(* IEC 61131-3 sources: PLC_02/HMI (part 2) *)

	IF (HMI.Rack4[13] AND 16#00ff) >= 1 AND (HMI.Rack4[13] AND 16#00ff) <= 164 THEN
		HMIBinding.CommonUI.sString5[0]		:= UINT_TO_STRING((HMI.Rack4[13] AND 16#00ff)) ;
	ELSIF (HMI.Rack4[13] AND 16#00ff) < 1 THEN
		HMIBinding.CommonUI.sString5[0]		:= '1';
	ELSE
		HMIBinding.CommonUI.sString5[0]		:= '164';
	END_IF;
	IF (HMI.Rack4[13]  /  16#0100) >= 1 AND (HMI.Rack4[13]  /  16#0100) <= 164 THEN
		HMIBinding.CommonUI.sString5[1] 		:= UINT_TO_STRING(HMI.Rack4[13]  /  16#0100) ;
	ELSIF (HMI.Rack4[13]  /  16#0100) < 1 THEN
		HMIBinding.CommonUI.sString5[1]		:= '1';
	ELSE
		HMIBinding.CommonUI.sString5[1]		:= '164';
	END_IF;
	HMIBinding.CommonUI.sString20[5]		:= CONCAT(HMIBinding.CommonUI.sString5[0],'(C)');
	HMIBinding.CommonUI.sString20[6]		:= CONCAT(HMIBinding.CommonUI.sString5[1],'(C)');

	IF (HMI.Rack4[14] AND 16#00ff) >= 1 AND (HMI.Rack4[14] AND 16#00ff) <= 164 THEN
		HMIBinding.CommonUI.sString5[0]		:= UINT_TO_STRING((HMI.Rack4[14] AND 16#00ff)) ;
	ELSIF (HMI.Rack4[14] AND 16#00ff) < 1 THEN
		HMIBinding.CommonUI.sString5[0]		:= '1';
	ELSE
		HMIBinding.CommonUI.sString5[0]		:= '164';
	END_IF;
	IF (HMI.Rack4[14]  /  16#0100) >= 1 AND (HMI.Rack4[14]  /  16#0100) <= 164 THEN
		HMIBinding.CommonUI.sString5[1] 		:= UINT_TO_STRING(HMI.Rack4[14]  /  16#0100) ;
	ELSIF (HMI.Rack4[14]  /  16#0100) < 1 THEN
		HMIBinding.CommonUI.sString5[1]		:= '1';
	ELSE
		HMIBinding.CommonUI.sString5[1]		:= '164';
	END_IF;
	HMIBinding.CommonUI.sString20[7]		:= CONCAT(HMIBinding.CommonUI.sString5[0],'(C)');
	HMIBinding.CommonUI.sString20[8]		:= CONCAT(HMIBinding.CommonUI.sString5[1],'(C)');

	IF HMI.Rack4[22] >= 672 AND HMI.Rack4[22] <= 1080 THEN
		HMIBinding.RackUI.sString5[0] 	:= REAL_TO_STRING(HMI.Rack4[22]*0.1) ;
	ELSIF HMI.Rack4[22] < 672 THEN
		HMIBinding.RackUI.sString5[0]	:= '67.2';
	ELSE
		HMIBinding.RackUI.sString5[0]	:= '108';
	END_IF;
	HMIBinding.RackUI.sString20[1]		:= CONCAT(HMIBinding.RackUI.sString5[0],'(V)');

	IF (HMI.Rack4[21].0) THEN
		HMIBinding.RackUI.sString20[0] := 'Solid_Green';
	ELSE
		HMIBinding.RackUI.sString20[0] := 'Solid_Red';
	END_IF;
	IF HMI.Rack4[23] >= 672 AND HMI.Rack4[23] <= 1080 THEN
		HMIBinding.RackUI.sString5[0] 	:= REAL_TO_STRING(HMI.Rack4[23]*0.1) ;
	ELSIF HMI.Rack4[23] < 672 THEN
		HMIBinding.RackUI.sString5[0]	:= '67.2';
	ELSE
		HMIBinding.RackUI.sString5[0]	:= '108';
	END_IF;
	HMIBinding.RackUI.sString20[3]		:= CONCAT(HMIBinding.RackUI.sString5[0],'(V)');

	IF (HMI.Rack4[21].1) THEN
		HMIBinding.RackUI.sString20[2] := 'Solid_Green';
	ELSE
		HMIBinding.RackUI.sString20[2] := 'Solid_Red';
	END_IF;

	IF HMI.Rack4[24] >= 672 AND HMI.Rack4[24] <= 1080 THEN
		HMIBinding.RackUI.sString5[0] 	:= REAL_TO_STRING(HMI.Rack4[24]*0.1) ;
	ELSIF HMI.Rack4[24] < 672 THEN
		HMIBinding.RackUI.sString5[0]	:= '67.2';
	ELSE
		HMIBinding.RackUI.sString5[0]	:= '108';
	END_IF;
	HMIBinding.RackUI.sString20[5]		:= CONCAT(HMIBinding.RackUI.sString5[0],'(V)');

	IF (HMI.Rack4[21].2) THEN
		HMIBinding.RackUI.sString20[4] := 'Solid_Green';
	ELSE
		HMIBinding.RackUI.sString20[4] := 'Solid_Red';
	END_IF;

	IF HMI.Rack4[25] >= 672 AND HMI.Rack4[25] <= 1080 THEN
		HMIBinding.RackUI.sString5[0] 	:= REAL_TO_STRING(HMI.Rack4[25]*0.1) ;
	ELSIF HMI.Rack4[25] < 672 THEN
		HMIBinding.RackUI.sString5[0]	:= '67.2';
	ELSE
		HMIBinding.RackUI.sString5[0]	:= '108';
	END_IF;
	HMIBinding.RackUI.sString20[7]		:= CONCAT(HMIBinding.RackUI.sString5[0],'(V)');

	IF (HMI.Rack4[21].3) THEN
		HMIBinding.RackUI.sString20[6] := 'Solid_Green';
	ELSE
		HMIBinding.RackUI.sString20[6] := 'Solid_Red';
	END_IF;
	IF HMI.Rack4[26] >= 672 AND HMI.Rack4[26] <= 1080 THEN
		HMIBinding.RackUI.sString5[0] 	:= REAL_TO_STRING(HMI.Rack4[26]*0.1) ;
	ELSIF HMI.Rack4[26] < 672 THEN
		HMIBinding.RackUI.sString5[0]	:= '67.2';
	ELSE
		HMIBinding.RackUI.sString5[0]	:= '108';
	END_IF;
	HMIBinding.RackUI.sString20[9]		:= CONCAT(HMIBinding.RackUI.sString5[0],'(V)');

	IF (HMI.Rack4[21].4) THEN
		HMIBinding.RackUI.sString20[8] := 'Solid_Green';
	ELSE
		HMIBinding.RackUI.sString20[8] := 'Solid_Red';
	END_IF;
	IF HMI.Rack4[27] >= 672 AND HMI.Rack4[27] <= 1080 THEN
		HMIBinding.RackUI.sString5[0] 	:= REAL_TO_STRING(HMI.Rack4[27]*0.1) ;
	ELSIF HMI.Rack4[27] < 672 THEN
		HMIBinding.RackUI.sString5[0]	:= '67.2';
	ELSE
		HMIBinding.RackUI.sString5[0]	:= '108';
	END_IF;
	HMIBinding.RackUI.sString20[11]		:= CONCAT(HMIBinding.RackUI.sString5[0],'(V)');

	IF (HMI.Rack4[21].5) THEN
		HMIBinding.RackUI.sString20[10] := 'Solid_Green';
	ELSE
		HMIBinding.RackUI.sString20[10] := 'Solid_Red';
	END_IF;
	IF HMI.Rack4[28] >= 672 AND HMI.Rack4[28] <= 1080 THEN
		HMIBinding.RackUI.sString5[0] 	:= REAL_TO_STRING(HMI.Rack4[28]*0.1) ;
	ELSIF HMI.Rack4[28] < 672 THEN
		HMIBinding.RackUI.sString5[0]	:= '67.2';
	ELSE
		HMIBinding.RackUI.sString5[0]	:= '108';
	END_IF;
	HMIBinding.RackUI.sString20[13]		:= CONCAT(HMIBinding.RackUI.sString5[0],'(V)');

	IF (HMI.Rack4[21].6) THEN
		HMIBinding.RackUI.sString20[12] := 'Solid_Green';
	ELSE
		HMIBinding.RackUI.sString20[12] := 'Solid_Red';
	END_IF;

	(* Over Current *)
	IF HMI.Rack4[17].0 THEN
		HMIBinding.RackUI.sString20[14] 		:= 'Solid_Red';
	ELSIF HMI.Rack4[16].0 THEN
		HMIBinding.RackUI.sString20[14]			:= 'Solid_Orange';
	ELSIF HMI.Rack4[15].0 THEN
		HMIBinding.RackUI.sString20[14]			:= 'Solid_Yellow';
	ELSE
		HMIBinding.RackUI.sString20[14]			:= 'Solid_Green';
	END_IF;

	(* Over SOC *)
	IF HMI.Rack4[17].1 THEN
		HMIBinding.RackUI.sString20[15]			:= 'Solid_Red';
	ELSIF HMI.Rack4[16].1 THEN
		HMIBinding.RackUI.sString20[15]			:= 'Solid_Orange';
	ELSIF HMI.Rack4[15].1 THEN
		HMIBinding.RackUI.sString20[15]			:= 'Solid_Yellow';
	ELSE
		HMIBinding.RackUI.sString20[15] 			:= 'Solid_Green';
	END_IF;

	(* Under SOC *)
	IF HMI.Rack4[17].2 THEN
		HMIBinding.RackUI.sString20[16] 			:= 'Solid_Red';
	ELSIF HMI.Rack4[16].2 THEN
		HMIBinding.RackUI.sString20[16]  			:= 'Solid_Orange';
	ELSIF HMI.Rack4[15].2 THEN
		HMIBinding.RackUI.sString20[16] 			:= 'Solid_Yellow';
	ELSE
		HMIBinding.RackUI.sString20[16]			:= 'Solid_Green';
	END_IF;

	(* Over Voltage *)
	IF HMI.Rack4[17].3 THEN
		HMIBinding.RackUI.sString20[17]			:= 'Solid_Red';
	ELSIF HMI.Rack4[16].3 THEN
		HMIBinding.RackUI.sString20[17] 			:= 'Solid_Orange';
	ELSIF HMI.Rack4[15].3 THEN
		HMIBinding.RackUI.sString20[17] 			:= 'Solid_Yellow';
	ELSE
		HMIBinding.RackUI.sString20[17] 			:= 'Solid_Green';
	END_IF;

	(* Under Voltage *)
	IF HMI.Rack4[17].4 THEN
		HMIBinding.RackUI.sString20[18] 			:= 'Solid_Red';
	ELSIF HMI.Rack4[16].4 THEN
		HMIBinding.RackUI.sString20[18] 			:= 'Solid_Orange';
	ELSIF HMI.Rack4[15].4 THEN
		HMIBinding.RackUI.sString20[18] 			:= 'Solid_Yellow';
	ELSE
		HMIBinding.RackUI.sString20[18] 			:= 'Solid_Green';
	END_IF;

	(* Cell Over Voltage *)
	IF HMI.Rack4[17].5 THEN
		HMIBinding.RackUI.sString20[19] 			:= 'Solid_Red';
	ELSIF HMI.Rack4[16].5 THEN
		HMIBinding.RackUI.sString20[19] 			:= 'Solid_Orange';
	ELSIF HMI.Rack4[15].5 THEN
		HMIBinding.RackUI.sString20[19] 			:= 'Solid_Yellow';
	ELSE
		HMIBinding.RackUI.sString20[19] 			:= 'Solid_Green';
	END_IF;

	(* Cell Under Voltage *)
	IF HMI.Rack4[17].6 THEN
		HMIBinding.RackUI.sString20[20] 			:= 'Solid_Red';
	ELSIF HMI.Rack4[16].6 THEN
		HMIBinding.RackUI.sString20[20] 			:= 'Solid_Orange';
	ELSIF HMI.Rack4[15].6 THEN
		HMIBinding.RackUI.sString20[20] 			:= 'Solid_Yellow';
	ELSE
		HMIBinding.RackUI.sString20[20] 			:= 'Solid_Green';
	END_IF;

	(* Cell UnBalance Voltage *)
	IF HMI.Rack4[17].7 THEN
		HMIBinding.RackUI.sString20[21]			:= 'Solid_Red';
	ELSIF HMI.Rack4[16].7 THEN
		HMIBinding.RackUI.sString20[21] 			:= 'Solid_Orange';
	ELSIF HMI.Rack4[15].7 THEN
		HMIBinding.RackUI.sString20[21]			:= 'Solid_Yellow';
	ELSE
		HMIBinding.RackUI.sString20[21]			:= 'Solid_Green';
	END_IF;

	(* Discahrger Cell Over Temperature *)
	IF HMI.Rack4[17].8 THEN
		HMIBinding.RackUI.sString20[22] 			:= 'Solid_Red';
	ELSIF HMI.Rack4[16].8 THEN
		HMIBinding.RackUI.sString20[22] 			:= 'Solid_Orange';
	ELSIF HMI.Rack4[15].8 THEN
		HMIBinding.RackUI.sString20[22] 			:= 'Solid_Yellow';
	ELSE
		HMIBinding.RackUI.sString20[22] 			:= 'Solid_Green';
	END_IF;

	(* Charger Cell Over Temperature *)
	IF HMI.Rack4[17].9 THEN
		HMIBinding.RackUI.sString20[23] 			:= 'Solid_Red';
	ELSIF HMI.Rack4[16].9 THEN
		HMIBinding.RackUI.sString20[23] 			:= 'Solid_Orange';
	ELSIF HMI.Rack4[15].9 THEN
		HMIBinding.RackUI.sString20[23] 			:= 'Solid_Yellow';
	ELSE
		HMIBinding.RackUI.sString20[23] 			:= 'Solid_Green';
	END_IF;

	(* Discahrger Cell Under Temperature *)
	IF HMI.Rack4[17].10 THEN
		HMIBinding.RackUI.sString20[24] 			:= 'Solid_Red';
	ELSIF HMI.Rack4[16].10 THEN
		HMIBinding.RackUI.sString20[24] 			:= 'Solid_Orange';
	ELSIF HMI.Rack4[15].10 THEN
		HMIBinding.RackUI.sString20[24] 			:= 'Solid_Yellow';
	ELSE
		HMIBinding.RackUI.sString20[24] 			:= 'Solid_Green';
	END_IF;

	(* Charger Cell Under Temperature *)
	IF HMI.Rack4[17].11 THEN
		HMIBinding.RackUI.sString20[25] 		:= 'Solid_Red';
	ELSIF HMI.Rack4[16].11 THEN
		HMIBinding.RackUI.sString20[25]			:= 'Solid_Orange';
	ELSIF HMI.Rack4[15].11 THEN
		HMIBinding.RackUI.sString20[25]			:= 'Solid_Yellow';
	ELSE
		HMIBinding.RackUI.sString20[25]			:= 'Solid_Green';
	END_IF;

	(* Cell UnBalance Temperature *)
	IF HMI.Rack4[17].12 THEN
		HMIBinding.RackUI.sString20[26] 		:= 'Solid_Red';
	ELSIF HMI.Rack4[16].12 THEN
		HMIBinding.RackUI.sString20[26]			:= 'Solid_Orange';
	ELSIF HMI.Rack4[15].12 THEN
		HMIBinding.RackUI.sString20[26]			:= 'Solid_Yellow';
	ELSE
		HMIBinding.RackUI.sString20[26]			:= 'Solid_Green';
	END_IF;

	(* Internal COM *)
	IF HMI.Rack4[17].15 THEN
		HMIBinding.RackUI.sString20[27] 		:= 'Solid_Red';
	ELSE
		HMIBinding.RackUI.sString20[27]			:= 'Solid_Green';
	END_IF;

	(* External COM *)
	IF HMI.Rack4[17].0 THEN
		HMIBinding.RackUI.sString20[28] 		:= 'Solid_Red';
	ELSE
		HMIBinding.RackUI.sString20[28]			:= 'Solid_Green';
	END_IF;

	(* RelayWelding *)
	IF HMI.Rack4[18].1 THEN
		HMIBinding.RackUI.sString20[29] 		:= 'Solid_Red';
	ELSE
		HMIBinding.RackUI.sString20[29]			:= 'Solid_Green';
	END_IF;

	(* WaterLeak *)
	IF HMI.Rack4[18].2 THEN
		HMIBinding.RackUI.sString20[30] 		:= 'Solid_Red';
	ELSE
		HMIBinding.RackUI.sString20[30]			:= 'Solid_Green';
	END_IF;

	(* InsulationRegister *)
	IF HMI.Rack4[18].3 THEN
		HMIBinding.RackUI.sString20[31] 		:= 'Solid_Red';
	ELSE
		HMIBinding.RackUI.sString20[31]			:= 'Solid_Green';
	END_IF;

	(* MDSFuse *)
	IF HMI.Rack4[18].4 THEN
		HMIBinding.RackUI.sString20[32] 		:= 'Solid_Red';
	ELSE
		HMIBinding.RackUI.sString20[32]			:= 'Solid_Green';
	END_IF;

	(* CoolingRack *)
	IF HMI.Rack4[18].5 THEN
		HMIBinding.RackUI.sString20[33] 		:= 'Solid_Red';
	ELSE
		HMIBinding.RackUI.sString20[33]			:= 'Solid_Green';
	END_IF;

	(* DIO *)
	IF HMI.Rack4[19].0 THEN
		HMIBinding.RackUI.sString20[34] 		:= 'Solid_Red';
	ELSE
		HMIBinding.RackUI.sString20[34]			:= 'Solid_Green';
	END_IF;
	IF HMI.Rack4[19].1 THEN
		HMIBinding.RackUI.sString20[35] 		:= 'Solid_Red';
	ELSE
		HMIBinding.RackUI.sString20[35]			:= 'Solid_Green';
	END_IF;
	IF HMI.Rack4[19].2 THEN
		HMIBinding.RackUI.sString20[36] 		:= 'Solid_Red';
	ELSE
		HMIBinding.RackUI.sString20[36]			:= 'Solid_Green';
	END_IF;
	IF HMI.Rack4[20].2 THEN
		HMIBinding.RackUI.sString20[37] 		:= 'Solid_Red';
	ELSE
		HMIBinding.RackUI.sString20[37]			:= 'Solid_Green';
	END_IF;
	IF HMI.Rack4[20].4 THEN
		HMIBinding.RackUI.sString20[38] 		:= 'Solid_Red';
	ELSE
		HMIBinding.RackUI.sString20[38]			:= 'Solid_Green';
	END_IF;
	IF HMI.Rack4[20].5 THEN
		HMIBinding.RackUI.sString20[39] 		:= 'Solid_Red';
	ELSE
		HMIBinding.RackUI.sString20[39]			:= 'Solid_Green';
	END_IF;
END_ACTION
ACTION AtRack5UI :

	CASE HMI.Rack5[0] OF
		0:  HMIBinding.CommonUI.sString20[0] := 'NONE';
		1:  HMIBinding.CommonUI.sString20[0] := 'STANDBY';
		2:  HMIBinding.CommonUI.sString20[0] := 'RUN';
		3:  HMIBinding.CommonUI.sString20[0] := 'ALARM';
		4:  HMIBinding.CommonUI.sString20[0] := 'FAULT';
		5:  HMIBinding.CommonUI.sString20[0] := 'PROTECT';
	END_CASE;

	IF HMI.Rack5[1] >= 4700 AND HMI.Rack5[1] <= 7140 THEN
		HMIBinding.CommonUI.rReal[0]		:= UINT_TO_REAL(HMI.Rack5[1]) * 0.1 ;
	ELSIF HMI.Rack5[1] < 4700 THEN
		HMIBinding.CommonUI.rReal[0]		:= 470.0;
	ELSE
		HMIBinding.CommonUI.rReal[0]		:= 714.0;
	END_IF;
	HMIBinding.CommonUI.sString20[1]		:= REAL_TO_STRING((HMIBinding.CommonUI.rReal[0]-400)*0.675);
	HMIBinding.CommonUI.sString50[0]		:= CONCAT('[{"select":"#gauge3","spin":[',CONCAT(HMIBinding.CommonUI.sString20[1],',0,0]}]'));

	IF UINT_TO_INT(HMI.Rack5[2]) >= -3000 AND UINT_TO_INT(HMI.Rack5[2]) <= 3000 THEN
		HMIBinding.CommonUI.rReal[1] 			:= (UINT_TO_REAL(HMI.Rack5[2]) * 0.1) ;
	ELSIF UINT_TO_INT(HMI.Rack5[2]) < -3000 THEN
		HMIBinding.CommonUI.rReal[1]			:= -300;
	ELSE
		HMIBinding.CommonUI.rReal[1]			:= 300;
	END_IF;
	HMIBinding.CommonUI.sString20[2]		:= REAL_TO_STRING(HMIBinding.CommonUI.rReal[1]*0.27+135);
	HMIBinding.CommonUI.sString50[1]		:= CONCAT('[{"select":"#gauge4","spin":[',CONCAT(HMIBinding.CommonUI.sString20[2],',0,0]}]'));

	IF UINT_TO_INT(HMI.Rack5[3]) >= -50 AND UINT_TO_INT(HMI.Rack5[3]) <= 1050 THEN
		HMIBinding.CommonUI.rReal[2]		:= UINT_TO_REAL(HMI.Rack5[3]) * 0.1 ;
	ELSIF UINT_TO_INT(HMI.Rack5[3]) < -50 THEN
		HMIBinding.CommonUI.rReal[2]		:= -5;
	ELSE
		HMIBinding.CommonUI.rReal[2]		:= 105;
	END_IF;
	HMIBinding.CommonUI.sString20[3]		:= REAL_TO_STRING(HMIBinding.CommonUI.rReal[2]*2.7);
	HMIBinding.CommonUI.sString50[2]		:= CONCAT('[{"select":"#gauge1","spin":[',CONCAT(HMIBinding.CommonUI.sString20[3],',0,0]}]'));

	IF HMI.Rack5[4] >= 750 AND HMI.Rack5[4] <= 1000 THEN
		HMIBinding.CommonUI.rReal[3]		:= UINT_TO_REAL(HMI.Rack5[4]) * 0.1 ;
	ELSIF HMI.Rack5[4] < 750 THEN
		HMIBinding.CommonUI.rReal[3]		:= 75;
	ELSE
		HMIBinding.CommonUI.rReal[3]		:= 100;
	END_IF;
	HMIBinding.CommonUI.sString20[4]		:= REAL_TO_STRING(HMIBinding.CommonUI.rReal[3]*2.7);
	HMIBinding.CommonUI.sString50[3]		:= CONCAT('[{"select":"#gauge2","spin":[',CONCAT(HMIBinding.CommonUI.sString20[4],',0,0]}]'));

	IF HMI.Rack5[5] >= 2000 AND HMI.Rack5[5] <= 4500 THEN
		HMIBinding.CommonUI.rReal[4] 		:= UINT_TO_REAL(HMI.Rack5[5]) * 0.001 ;
	ELSIF	HMI.Rack5[5] < 2000 THEN
		HMIBinding.CommonUI.rReal[4]		:= 2;
	ELSE
		HMIBinding.CommonUI.rReal[4]		:= 4.5;
	END_IF;
	IF HMI.Rack5[6] >= 2000 AND HMI.Rack5[6] <= 4500 THEN
		HMIBinding.CommonUI.rReal[5]		:= UINT_TO_REAL(HMI.Rack5[6]) * 0.001 ;
	ELSIF	HMI.Rack5[6] < 2000 THEN
		HMIBinding.CommonUI.rReal[5]		:= 2;
	ELSE
		HMIBinding.CommonUI.rReal[5]		:= 4.5;
	END_IF;
	IF HMI.Rack5[7] >= 2000 AND HMI.Rack5[7] <= 4500 THEN
		HMIBinding.CommonUI.rReal[6]		:= UINT_TO_REAL(HMI.Rack5[7]) * 0.001 ;
	ELSIF	HMI.Rack5[7] < 2000 THEN
		HMIBinding.CommonUI.rReal[6]		:= 2;
	ELSE
		HMIBinding.CommonUI.rReal[6]		:= 4.5;
	END_IF;
	IF HMI.Rack5[8] >= 0 AND HMI.Rack5[8] <= 500 THEN
		HMIBinding.CommonUI.rReal[7] 		:= UINT_TO_REAL(HMI.Rack5[8]) * 0.001 ;
	ELSE
		HMIBinding.CommonUI.rReal[7] 		:= 0.5;
	END_IF;
	IF UINT_TO_INT(HMI.Rack5[9]) >= -300 AND UINT_TO_INT(HMI.Rack5[9]) <= 1000 THEN
		HMIBinding.CommonUI.rReal[8] 		:= UINT_TO_REAL(HMI.Rack5[9]) * 0.1 ;
	ELSIF	UINT_TO_INT(HMI.Rack5[9]) < -300 THEN
		HMIBinding.CommonUI.rReal[8] 		:= -30;
	ELSE
		HMIBinding.CommonUI.rReal[8] 		:= 100;
	END_IF;
	IF UINT_TO_INT(HMI.Rack5[10]) >= -300 AND UINT_TO_INT(HMI.Rack5[10]) <= 1000 THEN
		HMIBinding.CommonUI.rReal[9]		:= UINT_TO_REAL(HMI.Rack5[10]) * 0.1 ;
	ELSIF	UINT_TO_INT(HMI.Rack5[10]) < -300 THEN
		HMIBinding.CommonUI.rReal[9]		:= -30;
	ELSE
		HMIBinding.CommonUI.rReal[9]		:= 100;
	END_IF;
	IF UINT_TO_INT(HMI.Rack5[11]) >= -300 AND UINT_TO_INT(HMI.Rack5[11]) <= 1000 THEN
		HMIBinding.CommonUI.rReal[10]		:= UINT_TO_REAL(HMI.Rack5[11]) * 0.1 ;
	ELSIF	UINT_TO_INT(HMI.Rack5[11]) < -300 THEN
		HMIBinding.CommonUI.rReal[10]		:= -30;
	ELSE
		HMIBinding.CommonUI.rReal[10]		:= 100;
	END_IF;
	IF HMI.Rack5[12] >= 0 AND HMI.Rack5[12] <= 100 THEN
		HMIBinding.CommonUI.rReal[11] 		:= UINT_TO_REAL(HMI.Rack5[12]) * 0.1 ;
	ELSE
		HMIBinding.CommonUI.rReal[11]		:= 10;
	END_IF;

	IF (HMI.Rack5[13] AND 16#00ff) >= 1 AND (HMI.Rack5[13] AND 16#00ff) <= 164 THEN
		HMIBinding.CommonUI.sString5[0]		:= UINT_TO_STRING((HMI.Rack5[13] AND 16#00ff)) ;
	ELSIF (HMI.Rack5[13] AND 16#00ff) < 1 THEN
		HMIBinding.CommonUI.sString5[0]		:= '1';
	ELSE
		HMIBinding.CommonUI.sString5[0]		:= '164';
	END_IF;
	IF (HMI.Rack5[13]  /  16#0100) >= 1 AND (HMI.Rack5[13]  /  16#0100) <= 164 THEN
		HMIBinding.CommonUI.sString5[1] 		:= UINT_TO_STRING(HMI.Rack5[13]  /  16#0100) ;
	ELSIF (HMI.Rack5[13]  /  16#0100) < 1 THEN
		HMIBinding.CommonUI.sString5[1]		:= '1';
	ELSE
		HMIBinding.CommonUI.sString5[1]		:= '164';
	END_IF;
	HMIBinding.CommonUI.sString20[5]		:= CONCAT(HMIBinding.CommonUI.sString5[0],'(C)');
	HMIBinding.CommonUI.sString20[6]		:= CONCAT(HMIBinding.CommonUI.sString5[1],'(C)');

	IF (HMI.Rack5[14] AND 16#00ff) >= 1 AND (HMI.Rack5[14] AND 16#00ff) <= 164 THEN
		HMIBinding.CommonUI.sString5[0]		:= UINT_TO_STRING((HMI.Rack5[14] AND 16#00ff)) ;
	ELSIF (HMI.Rack5[14] AND 16#00ff) < 1 THEN
		HMIBinding.CommonUI.sString5[0]		:= '1';
	ELSE
		HMIBinding.CommonUI.sString5[0]		:= '164';
	END_IF;
	IF (HMI.Rack5[14]  /  16#0100) >= 1 AND (HMI.Rack5[14]  /  16#0100) <= 164 THEN
		HMIBinding.CommonUI.sString5[1] 		:= UINT_TO_STRING(HMI.Rack5[14]  /  16#0100) ;
	ELSIF (HMI.Rack5[14]  /  16#0100) < 1 THEN
		HMIBinding.CommonUI.sString5[1]		:= '1';
	ELSE
		HMIBinding.CommonUI.sString5[1]		:= '164';
	END_IF;
	HMIBinding.CommonUI.sString20[7]		:= CONCAT(HMIBinding.CommonUI.sString5[0],'(C)');
	HMIBinding.CommonUI.sString20[8]		:= CONCAT(HMIBinding.CommonUI.sString5[1],'(C)');

	IF HMI.Rack5[22] >= 672 AND HMI.Rack5[22] <= 1080 THEN
		HMIBinding.RackUI.sString5[0] 	:= REAL_TO_STRING(HMI.Rack5[22]*0.1) ;
	ELSIF HMI.Rack5[22] < 672 THEN
		HMIBinding.RackUI.sString5[0]	:= '67.2';
	ELSE
		HMIBinding.RackUI.sString5[0]	:= '108';
	END_IF;
	HMIBinding.RackUI.sString20[1]		:= CONCAT(HMIBinding.RackUI.sString5[0],'(V)');

	IF (HMI.Rack5[21].0) THEN
		HMIBinding.RackUI.sString20[0] := 'Solid_Green';
	ELSE
		HMIBinding.RackUI.sString20[0] := 'Solid_Red';
	END_IF;
	IF HMI.Rack5[23] >= 672 AND HMI.Rack5[23] <= 1080 THEN
		HMIBinding.RackUI.sString5[0] 	:= REAL_TO_STRING(HMI.Rack5[23]*0.1) ;
	ELSIF HMI.Rack5[23] < 672 THEN
		HMIBinding.RackUI.sString5[0]	:= '67.2';
	ELSE
		HMIBinding.RackUI.sString5[0]	:= '108';
	END_IF;
	HMIBinding.RackUI.sString20[3]		:= CONCAT(HMIBinding.RackUI.sString5[0],'(V)');

	IF (HMI.Rack5[21].1) THEN
		HMIBinding.RackUI.sString20[2] := 'Solid_Green';
	ELSE
		HMIBinding.RackUI.sString20[2] := 'Solid_Red';
	END_IF;

	IF HMI.Rack5[24] >= 672 AND HMI.Rack5[24] <= 1080 THEN
		HMIBinding.RackUI.sString5[0] 	:= REAL_TO_STRING(HMI.Rack5[24]*0.1) ;
	ELSIF HMI.Rack5[24] < 672 THEN
		HMIBinding.RackUI.sString5[0]	:= '67.2';
	ELSE
		HMIBinding.RackUI.sString5[0]	:= '108';
	END_IF;
	HMIBinding.RackUI.sString20[5]		:= CONCAT(HMIBinding.RackUI.sString5[0],'(V)');

	IF (HMI.Rack5[21].2) THEN
		HMIBinding.RackUI.sString20[4] := 'Solid_Green';
	ELSE
		HMIBinding.RackUI.sString20[4] := 'Solid_Red';
	END_IF;

	IF HMI.Rack5[25] >= 672 AND HMI.Rack5[25] <= 1080 THEN
		HMIBinding.RackUI.sString5[0] 	:= REAL_TO_STRING(HMI.Rack5[25]*0.1) ;
	ELSIF HMI.Rack5[25] < 672 THEN
		HMIBinding.RackUI.sString5[0]	:= '67.2';
	ELSE
		HMIBinding.RackUI.sString5[0]	:= '108';
	END_IF;
	HMIBinding.RackUI.sString20[7]		:= CONCAT(HMIBinding.RackUI.sString5[0],'(V)');

	IF (HMI.Rack5[21].3) THEN
		HMIBinding.RackUI.sString20[6] := 'Solid_Green';
	ELSE
		HMIBinding.RackUI.sString20[6] := 'Solid_Red';
	END_IF;
	IF HMI.Rack5[26] >= 672 AND HMI.Rack5[26] <= 1080 THEN
		HMIBinding.RackUI.sString5[0] 	:= REAL_TO_STRING(HMI.Rack5[26]*0.1) ;
	ELSIF HMI.Rack5[26] < 672 THEN
		HMIBinding.RackUI.sString5[0]	:= '67.2';
	ELSE
		HMIBinding.RackUI.sString5[0]	:= '108';
	END_IF;
	HMIBinding.RackUI.sString20[9]		:= CONCAT(HMIBinding.RackUI.sString5[0],'(V)');

	IF (HMI.Rack5[21].4) THEN
		HMIBinding.RackUI.sString20[8] := 'Solid_Green';
	ELSE
		HMIBinding.RackUI.sString20[8] := 'Solid_Red';
	END_IF;
	IF HMI.Rack5[27] >= 672 AND HMI.Rack5[27] <= 1080 THEN
		HMIBinding.RackUI.sString5[0] 	:= REAL_TO_STRING(HMI.Rack5[27]*0.1) ;
	ELSIF HMI.Rack5[27] < 672 THEN
		HMIBinding.RackUI.sString5[0]	:= '67.2';
	ELSE
		HMIBinding.RackUI.sString5[0]	:= '108';
	END_IF;
	HMIBinding.RackUI.sString20[11]		:= CONCAT(HMIBinding.RackUI.sString5[0],'(V)');

	IF (HMI.Rack5[21].5) THEN
		HMIBinding.RackUI.sString20[10] := 'Solid_Green';
	ELSE
		HMIBinding.RackUI.sString20[10] := 'Solid_Red';
	END_IF;
	IF HMI.Rack5[28] >= 672 AND HMI.Rack5[28] <= 1080 THEN
		HMIBinding.RackUI.sString5[0] 	:= REAL_TO_STRING(HMI.Rack5[28]*0.1) ;
	ELSIF HMI.Rack5[28] < 672 THEN
		HMIBinding.RackUI.sString5[0]	:= '67.2';
	ELSE
		HMIBinding.RackUI.sString5[0]	:= '108';
	END_IF;
	HMIBinding.RackUI.sString20[13]		:= CONCAT(HMIBinding.RackUI.sString5[0],'(V)');

	IF (HMI.Rack5[21].6) THEN
		HMIBinding.RackUI.sString20[12] := 'Solid_Green';
	ELSE
		HMIBinding.RackUI.sString20[12] := 'Solid_Red';
	END_IF;

	(* Over Current *)
	IF HMI.Rack5[17].0 THEN
		HMIBinding.RackUI.sString20[14] 		:= 'Solid_Red';
	ELSIF HMI.Rack5[16].0 THEN
		HMIBinding.RackUI.sString20[14]			:= 'Solid_Orange';
	ELSIF HMI.Rack5[15].0 THEN
		HMIBinding.RackUI.sString20[14]			:= 'Solid_Yellow';
	ELSE
		HMIBinding.RackUI.sString20[14]			:= 'Solid_Green';
	END_IF;

	(* Over SOC *)
	IF HMI.Rack5[17].1 THEN
		HMIBinding.RackUI.sString20[15]			:= 'Solid_Red';
	ELSIF HMI.Rack5[16].1 THEN
		HMIBinding.RackUI.sString20[15]			:= 'Solid_Orange';
	ELSIF HMI.Rack5[15].1 THEN
		HMIBinding.RackUI.sString20[15]			:= 'Solid_Yellow';
	ELSE
		HMIBinding.RackUI.sString20[15] 			:= 'Solid_Green';
	END_IF;

	(* Under SOC *)
	IF HMI.Rack5[17].2 THEN
		HMIBinding.RackUI.sString20[16] 			:= 'Solid_Red';
	ELSIF HMI.Rack5[16].2 THEN
		HMIBinding.RackUI.sString20[16]  			:= 'Solid_Orange';
	ELSIF HMI.Rack5[15].2 THEN
		HMIBinding.RackUI.sString20[16] 			:= 'Solid_Yellow';
	ELSE
		HMIBinding.RackUI.sString20[16]			:= 'Solid_Green';
	END_IF;

	(* Over Voltage *)
	IF HMI.Rack5[17].3 THEN
		HMIBinding.RackUI.sString20[17]			:= 'Solid_Red';
	ELSIF HMI.Rack5[16].3 THEN
		HMIBinding.RackUI.sString20[17] 			:= 'Solid_Orange';
	ELSIF HMI.Rack5[15].3 THEN
		HMIBinding.RackUI.sString20[17] 			:= 'Solid_Yellow';
	ELSE
		HMIBinding.RackUI.sString20[17] 			:= 'Solid_Green';
	END_IF;

	(* Under Voltage *)
	IF HMI.Rack5[17].4 THEN
		HMIBinding.RackUI.sString20[18] 			:= 'Solid_Red';
	ELSIF HMI.Rack5[16].4 THEN
		HMIBinding.RackUI.sString20[18] 			:= 'Solid_Orange';
	ELSIF HMI.Rack5[15].4 THEN
		HMIBinding.RackUI.sString20[18] 			:= 'Solid_Yellow';
	ELSE
		HMIBinding.RackUI.sString20[18] 			:= 'Solid_Green';
	END_IF;

	(* Cell Over Voltage *)
	IF HMI.Rack5[17].5 THEN
		HMIBinding.RackUI.sString20[19] 			:= 'Solid_Red';
	ELSIF HMI.Rack5[16].5 THEN
		HMIBinding.RackUI.sString20[19] 			:= 'Solid_Orange';
	ELSIF HMI.Rack5[15].5 THEN
		HMIBinding.RackUI.sString20[19] 			:= 'Solid_Yellow';
	ELSE
		HMIBinding.RackUI.sString20[19] 			:= 'Solid_Green';
	END_IF;

	(* Cell Under Voltage *)
	IF HMI.Rack5[17].6 THEN
		HMIBinding.RackUI.sString20[20] 			:= 'Solid_Red';
	ELSIF HMI.Rack5[16].6 THEN
		HMIBinding.RackUI.sString20[20] 			:= 'Solid_Orange';
	ELSIF HMI.Rack5[15].6 THEN
		HMIBinding.RackUI.sString20[20] 			:= 'Solid_Yellow';
	ELSE
		HMIBinding.RackUI.sString20[20] 			:= 'Solid_Green';
	END_IF;

	(* Cell UnBalance Voltage *)
	IF HMI.Rack5[17].7 THEN
		HMIBinding.RackUI.sString20[21]			:= 'Solid_Red';
	ELSIF HMI.Rack5[16].7 THEN
		HMIBinding.RackUI.sString20[21] 			:= 'Solid_Orange';
	ELSIF HMI.Rack5[15].7 THEN
		HMIBinding.RackUI.sString20[21]			:= 'Solid_Yellow';
	ELSE
		HMIBinding.RackUI.sString20[21]			:= 'Solid_Green';
	END_IF;

	(* Discahrger Cell Over Temperature *)
	IF HMI.Rack5[17].8 THEN
		HMIBinding.RackUI.sString20[22] 			:= 'Solid_Red';
	ELSIF HMI.Rack5[16].8 THEN
		HMIBinding.RackUI.sString20[22] 			:= 'Solid_Orange';
	ELSIF HMI.Rack5[15].8 THEN
		HMIBinding.RackUI.sString20[22] 			:= 'Solid_Yellow';
	ELSE
		HMIBinding.RackUI.sString20[22] 			:= 'Solid_Green';
	END_IF;

	(* Charger Cell Over Temperature *)
	IF HMI.Rack5[17].9 THEN
		HMIBinding.RackUI.sString20[23] 			:= 'Solid_Red';
	ELSIF HMI.Rack5[16].9 THEN
		HMIBinding.RackUI.sString20[23] 			:= 'Solid_Orange';
	ELSIF HMI.Rack5[15].9 THEN
		HMIBinding.RackUI.sString20[23] 			:= 'Solid_Yellow';
	ELSE
		HMIBinding.RackUI.sString20[23] 			:= 'Solid_Green';
	END_IF;

	(* Discahrger Cell Under Temperature *)
	IF HMI.Rack5[17].10 THEN
		HMIBinding.RackUI.sString20[24] 			:= 'Solid_Red';
	ELSIF HMI.Rack5[16].10 THEN
		HMIBinding.RackUI.sString20[24] 			:= 'Solid_Orange';
	ELSIF HMI.Rack5[15].10 THEN
		HMIBinding.RackUI.sString20[24] 			:= 'Solid_Yellow';
	ELSE
		HMIBinding.RackUI.sString20[24] 			:= 'Solid_Green';
	END_IF;

	(* Charger Cell Under Temperature *)
	IF HMI.Rack5[17].11 THEN
		HMIBinding.RackUI.sString20[25] 		:= 'Solid_Red';
	ELSIF HMI.Rack5[16].11 THEN
		HMIBinding.RackUI.sString20[25]			:= 'Solid_Orange';
	ELSIF HMI.Rack5[15].11 THEN
		HMIBinding.RackUI.sString20[25]			:= 'Solid_Yellow';
	ELSE
		HMIBinding.RackUI.sString20[25]			:= 'Solid_Green';
	END_IF;

	(* Cell UnBalance Temperature *)
	IF HMI.Rack5[17].12 THEN
		HMIBinding.RackUI.sString20[26] 		:= 'Solid_Red';
	ELSIF HMI.Rack5[16].12 THEN
		HMIBinding.RackUI.sString20[26]			:= 'Solid_Orange';
	ELSIF HMI.Rack5[15].12 THEN
		HMIBinding.RackUI.sString20[26]			:= 'Solid_Yellow';
	ELSE
		HMIBinding.RackUI.sString20[26]			:= 'Solid_Green';
	END_IF;

	(* Internal COM *)
	IF HMI.Rack5[17].15 THEN
		HMIBinding.RackUI.sString20[27] 		:= 'Solid_Red';
	ELSE
		HMIBinding.RackUI.sString20[27]			:= 'Solid_Green';
	END_IF;

	(* External COM *)
	IF HMI.Rack5[17].0 THEN
		HMIBinding.RackUI.sString20[28] 		:= 'Solid_Red';
	ELSE
		HMIBinding.RackUI.sString20[28]			:= 'Solid_Green';
	END_IF;

	(* RelayWelding *)
	IF HMI.Rack5[18].1 THEN
		HMIBinding.RackUI.sString20[29] 		:= 'Solid_Red';
	ELSE
		HMIBinding.RackUI.sString20[29]			:= 'Solid_Green';
	END_IF;

	(* WaterLeak *)
	IF HMI.Rack5[18].2 THEN
		HMIBinding.RackUI.sString20[30] 		:= 'Solid_Red';
	ELSE
		HMIBinding.RackUI.sString20[30]			:= 'Solid_Green';
	END_IF;

	(* InsulationRegister *)
	IF HMI.Rack5[18].3 THEN
		HMIBinding.RackUI.sString20[31] 		:= 'Solid_Red';
	ELSE
		HMIBinding.RackUI.sString20[31]			:= 'Solid_Green';
	END_IF;

	(* MDSFuse *)
	IF HMI.Rack5[18].4 THEN
		HMIBinding.RackUI.sString20[32] 		:= 'Solid_Red';
	ELSE
		HMIBinding.RackUI.sString20[32]			:= 'Solid_Green';
	END_IF;

	(* CoolingRack *)
	IF HMI.Rack5[18].5 THEN
		HMIBinding.RackUI.sString20[33] 		:= 'Solid_Red';
	ELSE
		HMIBinding.RackUI.sString20[33]			:= 'Solid_Green';
	END_IF;

	(* DIO *)
	IF HMI.Rack5[19].0 THEN
		HMIBinding.RackUI.sString20[34] 		:= 'Solid_Red';
	ELSE
		HMIBinding.RackUI.sString20[34]			:= 'Solid_Green';
	END_IF;
	IF HMI.Rack5[19].1 THEN
		HMIBinding.RackUI.sString20[35] 		:= 'Solid_Red';
	ELSE
		HMIBinding.RackUI.sString20[35]			:= 'Solid_Green';
	END_IF;
	IF HMI.Rack5[19].2 THEN
		HMIBinding.RackUI.sString20[36] 		:= 'Solid_Red';
	ELSE
		HMIBinding.RackUI.sString20[36]			:= 'Solid_Green';
	END_IF;
	IF HMI.Rack5[20].2 THEN
		HMIBinding.RackUI.sString20[37] 		:= 'Solid_Red';
	ELSE
		HMIBinding.RackUI.sString20[37]			:= 'Solid_Green';
	END_IF;
	IF HMI.Rack5[20].4 THEN
		HMIBinding.RackUI.sString20[38] 		:= 'Solid_Red';
	ELSE
		HMIBinding.RackUI.sString20[38]			:= 'Solid_Green';
	END_IF;
	IF HMI.Rack5[20].5 THEN
		HMIBinding.RackUI.sString20[39] 		:= 'Solid_Red';
	ELSE
		HMIBinding.RackUI.sString20[39]			:= 'Solid_Green';
	END_IF;
END_ACTION
ACTION AtRack6UI :

	CASE HMI.Rack6[0] OF
		0:  HMIBinding.CommonUI.sString20[0] := 'NONE';
		1:  HMIBinding.CommonUI.sString20[0] := 'STANDBY';
		2:  HMIBinding.CommonUI.sString20[0] := 'RUN';
		3:  HMIBinding.CommonUI.sString20[0] := 'ALARM';
		4:  HMIBinding.CommonUI.sString20[0] := 'FAULT';
		5:  HMIBinding.CommonUI.sString20[0] := 'PROTECT';
	END_CASE;

	IF HMI.Rack6[1] >= 4700 AND HMI.Rack6[1] <= 7140 THEN
		HMIBinding.CommonUI.rReal[0]		:= UINT_TO_REAL(HMI.Rack6[1]) * 0.1 ;
	ELSIF HMI.Rack6[1] < 4700 THEN
		HMIBinding.CommonUI.rReal[0]		:= 470.0;
	ELSE
		HMIBinding.CommonUI.rReal[0]		:= 714.0;
	END_IF;
	HMIBinding.CommonUI.sString20[1]		:= REAL_TO_STRING((HMIBinding.CommonUI.rReal[0]-400)*0.675);
	HMIBinding.CommonUI.sString50[0]		:= CONCAT('[{"select":"#gauge3","spin":[',CONCAT(HMIBinding.CommonUI.sString20[1],',0,0]}]'));

	IF UINT_TO_INT(HMI.Rack6[2]) >= -3000 AND UINT_TO_INT(HMI.Rack6[2]) <= 3000 THEN
		HMIBinding.CommonUI.rReal[1] 			:= (UINT_TO_REAL(HMI.Rack6[2]) * 0.1) ;
	ELSIF UINT_TO_INT(HMI.Rack6[2]) < -3000 THEN
		HMIBinding.CommonUI.rReal[1]			:= -300;
	ELSE
		HMIBinding.CommonUI.rReal[1]			:= 300;
	END_IF;
	HMIBinding.CommonUI.sString20[2]		:= REAL_TO_STRING(HMIBinding.CommonUI.rReal[1]*0.27+135);
	HMIBinding.CommonUI.sString50[1]		:= CONCAT('[{"select":"#gauge4","spin":[',CONCAT(HMIBinding.CommonUI.sString20[2],',0,0]}]'));

	IF UINT_TO_INT(HMI.Rack6[3]) >= -50 AND UINT_TO_INT(HMI.Rack6[3]) <= 1050 THEN
		HMIBinding.CommonUI.rReal[2]		:= UINT_TO_REAL(HMI.Rack6[3]) * 0.1 ;
	ELSIF UINT_TO_INT(HMI.Rack6[3]) < -50 THEN
		HMIBinding.CommonUI.rReal[2]		:= -5;
	ELSE
		HMIBinding.CommonUI.rReal[2]		:= 105;
	END_IF;
	HMIBinding.CommonUI.sString20[3]		:= REAL_TO_STRING(HMIBinding.CommonUI.rReal[2]*2.7);
	HMIBinding.CommonUI.sString50[2]		:= CONCAT('[{"select":"#gauge1","spin":[',CONCAT(HMIBinding.CommonUI.sString20[3],',0,0]}]'));

	IF HMI.Rack6[4] >= 750 AND HMI.Rack6[4] <= 1000 THEN
		HMIBinding.CommonUI.rReal[3]		:= UINT_TO_REAL(HMI.Rack6[4]) * 0.1 ;
	ELSIF HMI.Rack6[4] < 750 THEN
		HMIBinding.CommonUI.rReal[3]		:= 75;
	ELSE
		HMIBinding.CommonUI.rReal[3]		:= 100;
	END_IF;
	HMIBinding.CommonUI.sString20[4]		:= REAL_TO_STRING(HMIBinding.CommonUI.rReal[3]*2.7);
	HMIBinding.CommonUI.sString50[3]		:= CONCAT('[{"select":"#gauge2","spin":[',CONCAT(HMIBinding.CommonUI.sString20[4],',0,0]}]'));

	IF HMI.Rack6[5] >= 2000 AND HMI.Rack6[5] <= 4500 THEN
		HMIBinding.CommonUI.rReal[4] 		:= UINT_TO_REAL(HMI.Rack6[5]) * 0.001 ;
	ELSIF	HMI.Rack6[5] < 2000 THEN
		HMIBinding.CommonUI.rReal[4]		:= 2;
	ELSE
		HMIBinding.CommonUI.rReal[4]		:= 4.5;
	END_IF;
	IF HMI.Rack6[6] >= 2000 AND HMI.Rack6[6] <= 4500 THEN
		HMIBinding.CommonUI.rReal[5]		:= UINT_TO_REAL(HMI.Rack6[6]) * 0.001 ;
	ELSIF	HMI.Rack6[6] < 2000 THEN
		HMIBinding.CommonUI.rReal[5]		:= 2;
	ELSE
		HMIBinding.CommonUI.rReal[5]		:= 4.5;
	END_IF;
	IF HMI.Rack6[7] >= 2000 AND HMI.Rack6[7] <= 4500 THEN
		HMIBinding.CommonUI.rReal[6]		:= UINT_TO_REAL(HMI.Rack6[7]) * 0.001 ;
	ELSIF	HMI.Rack6[7] < 2000 THEN
		HMIBinding.CommonUI.rReal[6]		:= 2;
	ELSE
		HMIBinding.CommonUI.rReal[6]		:= 4.5;
	END_IF;
	IF HMI.Rack6[8] >= 0 AND HMI.Rack6[8] <= 500 THEN
		HMIBinding.CommonUI.rReal[7] 		:= UINT_TO_REAL(HMI.Rack6[8]) * 0.001 ;
	ELSE
		HMIBinding.CommonUI.rReal[7] 		:= 0.5;
	END_IF;
	IF UINT_TO_INT(HMI.Rack6[9]) >= -300 AND UINT_TO_INT(HMI.Rack6[9]) <= 1000 THEN
		HMIBinding.CommonUI.rReal[8] 		:= UINT_TO_REAL(HMI.Rack6[9]) * 0.1 ;
	ELSIF	UINT_TO_INT(HMI.Rack6[9]) < -300 THEN
		HMIBinding.CommonUI.rReal[8] 		:= -30;
	ELSE
		HMIBinding.CommonUI.rReal[8] 		:= 100;
	END_IF;
	IF UINT_TO_INT(HMI.Rack6[10]) >= -300 AND UINT_TO_INT(HMI.Rack6[10]) <= 1000 THEN
		HMIBinding.CommonUI.rReal[9]		:= UINT_TO_REAL(HMI.Rack6[10]) * 0.1 ;
	ELSIF	UINT_TO_INT(HMI.Rack6[10]) < -300 THEN
		HMIBinding.CommonUI.rReal[9]		:= -30;
	ELSE
		HMIBinding.CommonUI.rReal[9]		:= 100;
	END_IF;
	IF UINT_TO_INT(HMI.Rack6[11]) >= -300 AND UINT_TO_INT(HMI.Rack6[11]) <= 1000 THEN
		HMIBinding.CommonUI.rReal[10]		:= UINT_TO_REAL(HMI.Rack6[11]) * 0.1 ;
	ELSIF	UINT_TO_INT(HMI.Rack6[11]) < -300 THEN
		HMIBinding.CommonUI.rReal[10]		:= -30;
	ELSE
		HMIBinding.CommonUI.rReal[10]		:= 100;
	END_IF;
	IF HMI.Rack6[12] >= 0 AND HMI.Rack6[12] <= 100 THEN
		HMIBinding.CommonUI.rReal[11] 		:= UINT_TO_REAL(HMI.Rack6[12]) * 0.1 ;
	ELSE
		HMIBinding.CommonUI.rReal[11]		:= 10;
	END_IF;

	IF (HMI.Rack6[13] AND 16#00ff) >= 1 AND (HMI.Rack6[13] AND 16#00ff) <= 164 THEN
		HMIBinding.CommonUI.sString5[0]		:= UINT_TO_STRING((HMI.Rack6[13] AND 16#00ff)) ;
	ELSIF (HMI.Rack6[13] AND 16#00ff) < 1 THEN
		HMIBinding.CommonUI.sString5[0]		:= '1';
	ELSE
		HMIBinding.CommonUI.sString5[0]		:= '164';
	END_IF;
	IF (HMI.Rack6[13]  /  16#0100) >= 1 AND (HMI.Rack6[13]  /  16#0100) <= 164 THEN
		HMIBinding.CommonUI.sString5[1] 		:= UINT_TO_STRING(HMI.Rack6[13]  /  16#0100) ;
	ELSIF (HMI.Rack6[13]  /  16#0100) < 1 THEN
		HMIBinding.CommonUI.sString5[1]		:= '1';
	ELSE
		HMIBinding.CommonUI.sString5[1]		:= '164';
	END_IF;
	HMIBinding.CommonUI.sString20[5]		:= CONCAT(HMIBinding.CommonUI.sString5[0],'(C)');
	HMIBinding.CommonUI.sString20[6]		:= CONCAT(HMIBinding.CommonUI.sString5[1],'(C)');

	IF (HMI.Rack6[14] AND 16#00ff) >= 1 AND (HMI.Rack6[14] AND 16#00ff) <= 164 THEN
		HMIBinding.CommonUI.sString5[0]		:= UINT_TO_STRING((HMI.Rack6[14] AND 16#00ff)) ;
	ELSIF (HMI.Rack6[14] AND 16#00ff) < 1 THEN
		HMIBinding.CommonUI.sString5[0]		:= '1';
	ELSE
		HMIBinding.CommonUI.sString5[0]		:= '164';
	END_IF;
	IF (HMI.Rack6[14]  /  16#0100) >= 1 AND (HMI.Rack6[14]  /  16#0100) <= 164 THEN
		HMIBinding.CommonUI.sString5[1] 		:= UINT_TO_STRING(HMI.Rack6[14]  /  16#0100) ;
	ELSIF (HMI.Rack6[14]  /  16#0100) < 1 THEN
		HMIBinding.CommonUI.sString5[1]		:= '1';
	ELSE
		HMIBinding.CommonUI.sString5[1]		:= '164';
	END_IF;
	HMIBinding.CommonUI.sString20[7]		:= CONCAT(HMIBinding.CommonUI.sString5[0],'(C)');
	HMIBinding.CommonUI.sString20[8]		:= CONCAT(HMIBinding.CommonUI.sString5[1],'(C)');

	IF HMI.Rack6[22] >= 672 AND HMI.Rack6[22] <= 1080 THEN
		HMIBinding.RackUI.sString5[0] 	:= REAL_TO_STRING(HMI.Rack6[22]*0.1) ;
	ELSIF HMI.Rack6[22] < 672 THEN
		HMIBinding.RackUI.sString5[0]	:= '67.2';
	ELSE
		HMIBinding.RackUI.sString5[0]	:= '108';
	END_IF;
	HMIBinding.RackUI.sString20[1]		:= CONCAT(HMIBinding.RackUI.sString5[0],'(V)');

	IF (HMI.Rack6[21].0) THEN
		HMIBinding.RackUI.sString20[0] := 'Solid_Green';
	ELSE
		HMIBinding.RackUI.sString20[0] := 'Solid_Red';
	END_IF;
	IF HMI.Rack6[23] >= 672 AND HMI.Rack6[23] <= 1080 THEN
		HMIBinding.RackUI.sString5[0] 	:= REAL_TO_STRING(HMI.Rack6[23]*0.1) ;
	ELSIF HMI.Rack6[23] < 672 THEN
		HMIBinding.RackUI.sString5[0]	:= '67.2';
	ELSE
		HMIBinding.RackUI.sString5[0]	:= '108';
	END_IF;
	HMIBinding.RackUI.sString20[3]		:= CONCAT(HMIBinding.RackUI.sString5[0],'(V)');

	IF (HMI.Rack6[21].1) THEN
		HMIBinding.RackUI.sString20[2] := 'Solid_Green';
	ELSE
		HMIBinding.RackUI.sString20[2] := 'Solid_Red';
	END_IF;

	IF HMI.Rack6[24] >= 672 AND HMI.Rack6[24] <= 1080 THEN
		HMIBinding.RackUI.sString5[0] 	:= REAL_TO_STRING(HMI.Rack6[24]*0.1) ;
	ELSIF HMI.Rack6[24] < 672 THEN
		HMIBinding.RackUI.sString5[0]	:= '67.2';
	ELSE
		HMIBinding.RackUI.sString5[0]	:= '108';
	END_IF;
	HMIBinding.RackUI.sString20[5]		:= CONCAT(HMIBinding.RackUI.sString5[0],'(V)');

	IF (HMI.Rack6[21].2) THEN
		HMIBinding.RackUI.sString20[4] := 'Solid_Green';
	ELSE
		HMIBinding.RackUI.sString20[4] := 'Solid_Red';
	END_IF;

	IF HMI.Rack6[25] >= 672 AND HMI.Rack6[25] <= 1080 THEN
		HMIBinding.RackUI.sString5[0] 	:= REAL_TO_STRING(HMI.Rack6[25]*0.1) ;
	ELSIF HMI.Rack6[25] < 672 THEN
		HMIBinding.RackUI.sString5[0]	:= '67.2';
	ELSE
		HMIBinding.RackUI.sString5[0]	:= '108';
	END_IF;
	HMIBinding.RackUI.sString20[7]		:= CONCAT(HMIBinding.RackUI.sString5[0],'(V)');

	IF (HMI.Rack6[21].3) THEN
		HMIBinding.RackUI.sString20[6] := 'Solid_Green';
	ELSE
		HMIBinding.RackUI.sString20[6] := 'Solid_Red';
	END_IF;
	IF HMI.Rack6[26] >= 672 AND HMI.Rack6[26] <= 1080 THEN
		HMIBinding.RackUI.sString5[0] 	:= REAL_TO_STRING(HMI.Rack6[26]*0.1) ;
	ELSIF HMI.Rack6[26] < 672 THEN
		HMIBinding.RackUI.sString5[0]	:= '67.2';
	ELSE
		HMIBinding.RackUI.sString5[0]	:= '108';
	END_IF;
	HMIBinding.RackUI.sString20[9]		:= CONCAT(HMIBinding.RackUI.sString5[0],'(V)');

	IF (HMI.Rack6[21].4) THEN
		HMIBinding.RackUI.sString20[8] := 'Solid_Green';
	ELSE
		HMIBinding.RackUI.sString20[8] := 'Solid_Red';
	END_IF;
	IF HMI.Rack6[27] >= 672 AND HMI.Rack6[27] <= 1080 THEN
		HMIBinding.RackUI.sString5[0] 	:= REAL_TO_STRING(HMI.Rack6[27]*0.1) ;
	ELSIF HMI.Rack6[27] < 672 THEN
		HMIBinding.RackUI.sString5[0]	:= '67.2';
	ELSE
		HMIBinding.RackUI.sString5[0]	:= '108';
	END_IF;
	HMIBinding.RackUI.sString20[11]		:= CONCAT(HMIBinding.RackUI.sString5[0],'(V)');

	IF (HMI.Rack6[21].5) THEN
		HMIBinding.RackUI.sString20[10] := 'Solid_Green';
	ELSE
		HMIBinding.RackUI.sString20[10] := 'Solid_Red';
	END_IF;
	IF HMI.Rack6[28] >= 672 AND HMI.Rack6[28] <= 1080 THEN
		HMIBinding.RackUI.sString5[0] 	:= REAL_TO_STRING(HMI.Rack6[28]*0.1) ;
	ELSIF HMI.Rack6[28] < 672 THEN
		HMIBinding.RackUI.sString5[0]	:= '67.2';
	ELSE
		HMIBinding.RackUI.sString5[0]	:= '108';
	END_IF;
	HMIBinding.RackUI.sString20[13]		:= CONCAT(HMIBinding.RackUI.sString5[0],'(V)');

	IF (HMI.Rack6[21].6) THEN
		HMIBinding.RackUI.sString20[12] := 'Solid_Green';
	ELSE
		HMIBinding.RackUI.sString20[12] := 'Solid_Red';
	END_IF;

	(* Over Current *)
	IF HMI.Rack6[17].0 THEN
		HMIBinding.RackUI.sString20[14] 		:= 'Solid_Red';
	ELSIF HMI.Rack6[16].0 THEN
		HMIBinding.RackUI.sString20[14]			:= 'Solid_Orange';
	ELSIF HMI.Rack6[15].0 THEN
		HMIBinding.RackUI.sString20[14]			:= 'Solid_Yellow';
	ELSE
		HMIBinding.RackUI.sString20[14]			:= 'Solid_Green';
	END_IF;

	(* Over SOC *)
	IF HMI.Rack6[17].1 THEN
		HMIBinding.RackUI.sString20[15]			:= 'Solid_Red';
	ELSIF HMI.Rack6[16].1 THEN
		HMIBinding.RackUI.sString20[15]			:= 'Solid_Orange';
	ELSIF HMI.Rack6[15].1 THEN
		HMIBinding.RackUI.sString20[15]			:= 'Solid_Yellow';
	ELSE
		HMIBinding.RackUI.sString20[15] 			:= 'Solid_Green';
	END_IF;

	(* Under SOC *)
	IF HMI.Rack6[17].2 THEN
		HMIBinding.RackUI.sString20[16] 			:= 'Solid_Red';
	ELSIF HMI.Rack6[16].2 THEN
		HMIBinding.RackUI.sString20[16]  			:= 'Solid_Orange';
	ELSIF HMI.Rack6[15].2 THEN
		HMIBinding.RackUI.sString20[16] 			:= 'Solid_Yellow';
	ELSE
		HMIBinding.RackUI.sString20[16]			:= 'Solid_Green';
	END_IF;

	(* Over Voltage *)
	IF HMI.Rack6[17].3 THEN
		HMIBinding.RackUI.sString20[17]			:= 'Solid_Red';
	ELSIF HMI.Rack6[16].3 THEN
		HMIBinding.RackUI.sString20[17] 			:= 'Solid_Orange';
	ELSIF HMI.Rack6[15].3 THEN
		HMIBinding.RackUI.sString20[17] 			:= 'Solid_Yellow';
	ELSE
		HMIBinding.RackUI.sString20[17] 			:= 'Solid_Green';
	END_IF;

	(* Under Voltage *)
	IF HMI.Rack6[17].4 THEN
		HMIBinding.RackUI.sString20[18] 			:= 'Solid_Red';
	ELSIF HMI.Rack6[16].4 THEN
		HMIBinding.RackUI.sString20[18] 			:= 'Solid_Orange';
	ELSIF HMI.Rack6[15].4 THEN
		HMIBinding.RackUI.sString20[18] 			:= 'Solid_Yellow';
	ELSE
		HMIBinding.RackUI.sString20[18] 			:= 'Solid_Green';
	END_IF;

	(* Cell Over Voltage *)
	IF HMI.Rack6[17].5 THEN
		HMIBinding.RackUI.sString20[19] 			:= 'Solid_Red';
	ELSIF HMI.Rack6[16].5 THEN
		HMIBinding.RackUI.sString20[19] 			:= 'Solid_Orange';
	ELSIF HMI.Rack6[15].5 THEN
		HMIBinding.RackUI.sString20[19] 			:= 'Solid_Yellow';
	ELSE
		HMIBinding.RackUI.sString20[19] 			:= 'Solid_Green';
	END_IF;

	(* Cell Under Voltage *)
	IF HMI.Rack6[17].6 THEN
		HMIBinding.RackUI.sString20[20] 			:= 'Solid_Red';
	ELSIF HMI.Rack6[16].6 THEN
		HMIBinding.RackUI.sString20[20] 			:= 'Solid_Orange';
	ELSIF HMI.Rack6[15].6 THEN
		HMIBinding.RackUI.sString20[20] 			:= 'Solid_Yellow';
	ELSE
		HMIBinding.RackUI.sString20[20] 			:= 'Solid_Green';
	END_IF;

	(* Cell UnBalance Voltage *)
	IF HMI.Rack6[17].7 THEN
		HMIBinding.RackUI.sString20[21]			:= 'Solid_Red';
	ELSIF HMI.Rack6[16].7 THEN
		HMIBinding.RackUI.sString20[21] 			:= 'Solid_Orange';
	ELSIF HMI.Rack6[15].7 THEN
		HMIBinding.RackUI.sString20[21]			:= 'Solid_Yellow';
	ELSE
		HMIBinding.RackUI.sString20[21]			:= 'Solid_Green';
	END_IF;

	(* Discahrger Cell Over Temperature *)
	IF HMI.Rack6[17].8 THEN
		HMIBinding.RackUI.sString20[22] 			:= 'Solid_Red';
	ELSIF HMI.Rack6[16].8 THEN
		HMIBinding.RackUI.sString20[22] 			:= 'Solid_Orange';
	ELSIF HMI.Rack6[15].8 THEN
		HMIBinding.RackUI.sString20[22] 			:= 'Solid_Yellow';
	ELSE
		HMIBinding.RackUI.sString20[22] 			:= 'Solid_Green';
	END_IF;

	(* Charger Cell Over Temperature *)
	IF HMI.Rack6[17].9 THEN
		HMIBinding.RackUI.sString20[23] 			:= 'Solid_Red';
	ELSIF HMI.Rack6[16].9 THEN
		HMIBinding.RackUI.sString20[23] 			:= 'Solid_Orange';
	ELSIF HMI.Rack6[15].9 THEN
		HMIBinding.RackUI.sString20[23] 			:= 'Solid_Yellow';
	ELSE
		HMIBinding.RackUI.sString20[23] 			:= 'Solid_Green';
	END_IF;

	(* Discahrger Cell Under Temperature *)
	IF HMI.Rack6[17].10 THEN
		HMIBinding.RackUI.sString20[24] 			:= 'Solid_Red';
	ELSIF HMI.Rack6[16].10 THEN
		HMIBinding.RackUI.sString20[24] 			:= 'Solid_Orange';
	ELSIF HMI.Rack6[15].10 THEN
		HMIBinding.RackUI.sString20[24] 			:= 'Solid_Yellow';
	ELSE
		HMIBinding.RackUI.sString20[24] 			:= 'Solid_Green';
	END_IF;

	(* Charger Cell Under Temperature *)
	IF HMI.Rack6[17].11 THEN
		HMIBinding.RackUI.sString20[25] 		:= 'Solid_Red';
	ELSIF HMI.Rack6[16].11 THEN
		HMIBinding.RackUI.sString20[25]			:= 'Solid_Orange';
	ELSIF HMI.Rack6[15].11 THEN
		HMIBinding.RackUI.sString20[25]			:= 'Solid_Yellow';
	ELSE
		HMIBinding.RackUI.sString20[25]			:= 'Solid_Green';
	END_IF;

	(* Cell UnBalance Temperature *)
	IF HMI.Rack6[17].12 THEN
		HMIBinding.RackUI.sString20[26] 		:= 'Solid_Red';
	ELSIF HMI.Rack6[16].12 THEN
		HMIBinding.RackUI.sString20[26]			:= 'Solid_Orange';
	ELSIF HMI.Rack6[15].12 THEN
		HMIBinding.RackUI.sString20[26]			:= 'Solid_Yellow';
	ELSE
		HMIBinding.RackUI.sString20[26]			:= 'Solid_Green';
	END_IF;

	(* Internal COM *)
	IF HMI.Rack6[17].15 THEN
		HMIBinding.RackUI.sString20[27] 		:= 'Solid_Red';
	ELSE
		HMIBinding.RackUI.sString20[27]			:= 'Solid_Green';
	END_IF;

	(* External COM *)
	IF HMI.Rack6[17].0 THEN
		HMIBinding.RackUI.sString20[28] 		:= 'Solid_Red';
	ELSE
		HMIBinding.RackUI.sString20[28]			:= 'Solid_Green';
	END_IF;

	(* RelayWelding *)
	IF HMI.Rack6[18].1 THEN
		HMIBinding.RackUI.sString20[29] 		:= 'Solid_Red';
	ELSE
		HMIBinding.RackUI.sString20[29]			:= 'Solid_Green';
	END_IF;

	(* WaterLeak *)
	IF HMI.Rack6[18].2 THEN
		HMIBinding.RackUI.sString20[30] 		:= 'Solid_Red';
	ELSE
		HMIBinding.RackUI.sString20[30]			:= 'Solid_Green';
	END_IF;

	(* InsulationRegister *)
	IF HMI.Rack6[18].3 THEN
		HMIBinding.RackUI.sString20[31] 		:= 'Solid_Red';
	ELSE
		HMIBinding.RackUI.sString20[31]			:= 'Solid_Green';
	END_IF;

	(* MDSFuse *)
	IF HMI.Rack6[18].4 THEN
		HMIBinding.RackUI.sString20[32] 		:= 'Solid_Red';
	ELSE
		HMIBinding.RackUI.sString20[32]			:= 'Solid_Green';
	END_IF;

	(* CoolingRack *)
	IF HMI.Rack6[18].5 THEN
		HMIBinding.RackUI.sString20[33] 		:= 'Solid_Red';
	ELSE
		HMIBinding.RackUI.sString20[33]			:= 'Solid_Green';
	END_IF;

	(* DIO *)
	IF HMI.Rack6[19].0 THEN
		HMIBinding.RackUI.sString20[34] 		:= 'Solid_Red';
	ELSE
		HMIBinding.RackUI.sString20[34]			:= 'Solid_Green';
	END_IF;
	IF HMI.Rack6[19].1 THEN
		HMIBinding.RackUI.sString20[35] 		:= 'Solid_Red';
	ELSE
		HMIBinding.RackUI.sString20[35]			:= 'Solid_Green';
	END_IF;
	IF HMI.Rack6[19].2 THEN
		HMIBinding.RackUI.sString20[36] 		:= 'Solid_Red';
	ELSE
		HMIBinding.RackUI.sString20[36]			:= 'Solid_Green';
	END_IF;
	IF HMI.Rack6[20].2 THEN
		HMIBinding.RackUI.sString20[37] 		:= 'Solid_Red';
	ELSE
		HMIBinding.RackUI.sString20[37]			:= 'Solid_Green';
	END_IF;
	IF HMI.Rack6[20].4 THEN
		HMIBinding.RackUI.sString20[38] 		:= 'Solid_Red';
	ELSE
		HMIBinding.RackUI.sString20[38]			:= 'Solid_Green';
	END_IF;
	IF HMI.Rack6[20].5 THEN
		HMIBinding.RackUI.sString20[39] 		:= 'Solid_Red';
	ELSE
		HMIBinding.RackUI.sString20[39]			:= 'Solid_Green';
	END_IF;
END_ACTION
ACTION AtRack7UI :

	CASE HMI.Rack7[0] OF
		0:  HMIBinding.CommonUI.sString20[0] := 'NONE';
		1:  HMIBinding.CommonUI.sString20[0] := 'STANDBY';
		2:  HMIBinding.CommonUI.sString20[0] := 'RUN';
		3:  HMIBinding.CommonUI.sString20[0] := 'ALARM';
		4:  HMIBinding.CommonUI.sString20[0] := 'FAULT';
		5:  HMIBinding.CommonUI.sString20[0] := 'PROTECT';
	END_CASE;

	IF HMI.Rack7[1] >= 4700 AND HMI.Rack7[1] <= 7140 THEN
		HMIBinding.CommonUI.rReal[0]		:= UINT_TO_REAL(HMI.Rack7[1]) * 0.1 ;
	ELSIF HMI.Rack7[1] < 4700 THEN
		HMIBinding.CommonUI.rReal[0]		:= 470.0;
	ELSE
		HMIBinding.CommonUI.rReal[0]		:= 714.0;
	END_IF;
	HMIBinding.CommonUI.sString20[1]		:= REAL_TO_STRING((HMIBinding.CommonUI.rReal[0]-400)*0.675);
	HMIBinding.CommonUI.sString50[0]		:= CONCAT('[{"select":"#gauge3","spin":[',CONCAT(HMIBinding.CommonUI.sString20[1],',0,0]}]'));

	IF UINT_TO_INT(HMI.Rack7[2]) >= -3000 AND UINT_TO_INT(HMI.Rack7[2]) <= 3000 THEN
		HMIBinding.CommonUI.rReal[1] 			:= (UINT_TO_REAL(HMI.Rack7[2]) * 0.1) ;
	ELSIF UINT_TO_INT(HMI.Rack7[2]) < -3000 THEN
		HMIBinding.CommonUI.rReal[1]			:= -300;
	ELSE
		HMIBinding.CommonUI.rReal[1]			:= 300;
	END_IF;
	HMIBinding.CommonUI.sString20[2]		:= REAL_TO_STRING(HMIBinding.CommonUI.rReal[1]*0.27+135);
	HMIBinding.CommonUI.sString50[1]		:= CONCAT('[{"select":"#gauge4","spin":[',CONCAT(HMIBinding.CommonUI.sString20[2],',0,0]}]'));

	IF UINT_TO_INT(HMI.Rack7[3]) >= -50 AND UINT_TO_INT(HMI.Rack7[3]) <= 1050 THEN
		HMIBinding.CommonUI.rReal[2]		:= UINT_TO_REAL(HMI.Rack7[3]) * 0.1 ;
	ELSIF UINT_TO_INT(HMI.Rack7[3]) < -50 THEN
		HMIBinding.CommonUI.rReal[2]		:= -5;
	ELSE
		HMIBinding.CommonUI.rReal[2]		:= 105;
	END_IF;
	HMIBinding.CommonUI.sString20[3]		:= REAL_TO_STRING(HMIBinding.CommonUI.rReal[2]*2.7);
	HMIBinding.CommonUI.sString50[2]		:= CONCAT('[{"select":"#gauge1","spin":[',CONCAT(HMIBinding.CommonUI.sString20[3],',0,0]}]'));

	IF HMI.Rack7[4] >= 750 AND HMI.Rack7[4] <= 1000 THEN
		HMIBinding.CommonUI.rReal[3]		:= UINT_TO_REAL(HMI.Rack7[4]) * 0.1 ;
	ELSIF HMI.Rack7[4] < 750 THEN
		HMIBinding.CommonUI.rReal[3]		:= 75;
	ELSE
		HMIBinding.CommonUI.rReal[3]		:= 100;
	END_IF;
	HMIBinding.CommonUI.sString20[4]		:= REAL_TO_STRING(HMIBinding.CommonUI.rReal[3]*2.7);
	HMIBinding.CommonUI.sString50[3]		:= CONCAT('[{"select":"#gauge2","spin":[',CONCAT(HMIBinding.CommonUI.sString20[4],',0,0]}]'));

	IF HMI.Rack7[5] >= 2000 AND HMI.Rack7[5] <= 4500 THEN
		HMIBinding.CommonUI.rReal[4] 		:= UINT_TO_REAL(HMI.Rack7[5]) * 0.001 ;
	ELSIF	HMI.Rack7[5] < 2000 THEN
		HMIBinding.CommonUI.rReal[4]		:= 2;
	ELSE
		HMIBinding.CommonUI.rReal[4]		:= 4.5;
	END_IF;
	IF HMI.Rack7[6] >= 2000 AND HMI.Rack7[6] <= 4500 THEN
		HMIBinding.CommonUI.rReal[5]		:= UINT_TO_REAL(HMI.Rack7[6]) * 0.001 ;
	ELSIF	HMI.Rack7[6] < 2000 THEN
		HMIBinding.CommonUI.rReal[5]		:= 2;
	ELSE
		HMIBinding.CommonUI.rReal[5]		:= 4.5;
	END_IF;
	IF HMI.Rack7[7] >= 2000 AND HMI.Rack7[7] <= 4500 THEN
		HMIBinding.CommonUI.rReal[6]		:= UINT_TO_REAL(HMI.Rack7[7]) * 0.001 ;
	ELSIF	HMI.Rack7[7] < 2000 THEN
		HMIBinding.CommonUI.rReal[6]		:= 2;
	ELSE
		HMIBinding.CommonUI.rReal[6]		:= 4.5;
	END_IF;
	IF HMI.Rack7[8] >= 0 AND HMI.Rack7[8] <= 500 THEN
		HMIBinding.CommonUI.rReal[7] 		:= UINT_TO_REAL(HMI.Rack7[8]) * 0.001 ;
	ELSE
		HMIBinding.CommonUI.rReal[7] 		:= 0.5;
	END_IF;
	IF UINT_TO_INT(HMI.Rack7[9]) >= -300 AND UINT_TO_INT(HMI.Rack7[9]) <= 1000 THEN
		HMIBinding.CommonUI.rReal[8] 		:= UINT_TO_REAL(HMI.Rack7[9]) * 0.1 ;
	ELSIF	UINT_TO_INT(HMI.Rack7[9]) < -300 THEN
		HMIBinding.CommonUI.rReal[8] 		:= -30;
	ELSE
		HMIBinding.CommonUI.rReal[8] 		:= 100;
	END_IF;
	IF UINT_TO_INT(HMI.Rack7[10]) >= -300 AND UINT_TO_INT(HMI.Rack7[10]) <= 1000 THEN
		HMIBinding.CommonUI.rReal[9]		:= UINT_TO_REAL(HMI.Rack7[10]) * 0.1 ;
	ELSIF	UINT_TO_INT(HMI.Rack7[10]) < -300 THEN
		HMIBinding.CommonUI.rReal[9]		:= -30;
	ELSE
		HMIBinding.CommonUI.rReal[9]		:= 100;
	END_IF;
	IF UINT_TO_INT(HMI.Rack7[11]) >= -300 AND UINT_TO_INT(HMI.Rack7[11]) <= 1000 THEN
		HMIBinding.CommonUI.rReal[10]		:= UINT_TO_REAL(HMI.Rack7[11]) * 0.1 ;
	ELSIF	UINT_TO_INT(HMI.Rack7[11]) < -300 THEN
		HMIBinding.CommonUI.rReal[10]		:= -30;
	ELSE
		HMIBinding.CommonUI.rReal[10]		:= 100;
	END_IF;
	IF HMI.Rack7[12] >= 0 AND HMI.Rack7[12] <= 100 THEN
		HMIBinding.CommonUI.rReal[11] 		:= UINT_TO_REAL(HMI.Rack7[12]) * 0.1 ;
	ELSE
		HMIBinding.CommonUI.rReal[11]		:= 10;
	END_IF;

	IF (HMI.Rack7[13] AND 16#00ff) >= 1 AND (HMI.Rack7[13] AND 16#00ff) <= 164 THEN
		HMIBinding.CommonUI.sString5[0]		:= UINT_TO_STRING((HMI.Rack7[13] AND 16#00ff)) ;
	ELSIF (HMI.Rack7[13] AND 16#00ff) < 1 THEN
		HMIBinding.CommonUI.sString5[0]		:= '1';
	ELSE
		HMIBinding.CommonUI.sString5[0]		:= '164';
	END_IF;
	IF (HMI.Rack7[13]  /  16#0100) >= 1 AND (HMI.Rack7[13]  /  16#0100) <= 164 THEN
		HMIBinding.CommonUI.sString5[1] 		:= UINT_TO_STRING(HMI.Rack7[13]  /  16#0100) ;
	ELSIF (HMI.Rack7[13]  /  16#0100) < 1 THEN
		HMIBinding.CommonUI.sString5[1]		:= '1';
	ELSE
		HMIBinding.CommonUI.sString5[1]		:= '164';
	END_IF;
	HMIBinding.CommonUI.sString20[5]		:= CONCAT(HMIBinding.CommonUI.sString5[0],'(C)');
	HMIBinding.CommonUI.sString20[6]		:= CONCAT(HMIBinding.CommonUI.sString5[1],'(C)');

	IF (HMI.Rack7[14] AND 16#00ff) >= 1 AND (HMI.Rack7[14] AND 16#00ff) <= 164 THEN
		HMIBinding.CommonUI.sString5[0]		:= UINT_TO_STRING((HMI.Rack7[14] AND 16#00ff)) ;
	ELSIF (HMI.Rack7[14] AND 16#00ff) < 1 THEN
		HMIBinding.CommonUI.sString5[0]		:= '1';
	ELSE
		HMIBinding.CommonUI.sString5[0]		:= '164';
	END_IF;
	IF (HMI.Rack7[14]  /  16#0100) >= 1 AND (HMI.Rack7[14]  /  16#0100) <= 164 THEN
		HMIBinding.CommonUI.sString5[1] 		:= UINT_TO_STRING(HMI.Rack7[14]  /  16#0100) ;
	ELSIF (HMI.Rack7[14]  /  16#0100) < 1 THEN
		HMIBinding.CommonUI.sString5[1]		:= '1';
	ELSE
		HMIBinding.CommonUI.sString5[1]		:= '164';
	END_IF;
	HMIBinding.CommonUI.sString20[7]		:= CONCAT(HMIBinding.CommonUI.sString5[0],'(C)');
	HMIBinding.CommonUI.sString20[8]		:= CONCAT(HMIBinding.CommonUI.sString5[1],'(C)');

	IF HMI.Rack7[22] >= 672 AND HMI.Rack7[22] <= 1080 THEN
		HMIBinding.RackUI.sString5[0] 	:= REAL_TO_STRING(HMI.Rack7[22]*0.1) ;
	ELSIF HMI.Rack7[22] < 672 THEN
		HMIBinding.RackUI.sString5[0]	:= '67.2';
	ELSE
		HMIBinding.RackUI.sString5[0]	:= '108';
	END_IF;
	HMIBinding.RackUI.sString20[1]		:= CONCAT(HMIBinding.RackUI.sString5[0],'(V)');

	IF (HMI.Rack7[21].0) THEN
		HMIBinding.RackUI.sString20[0] := 'Solid_Green';
	ELSE
		HMIBinding.RackUI.sString20[0] := 'Solid_Red';
	END_IF;
	IF HMI.Rack7[23] >= 672 AND HMI.Rack7[23] <= 1080 THEN
		HMIBinding.RackUI.sString5[0] 	:= REAL_TO_STRING(HMI.Rack7[23]*0.1) ;
	ELSIF HMI.Rack7[23] < 672 THEN
		HMIBinding.RackUI.sString5[0]	:= '67.2';
	ELSE
		HMIBinding.RackUI.sString5[0]	:= '108';
	END_IF;
	HMIBinding.RackUI.sString20[3]		:= CONCAT(HMIBinding.RackUI.sString5[0],'(V)');

	IF (HMI.Rack7[21].1) THEN
		HMIBinding.RackUI.sString20[2] := 'Solid_Green';
	ELSE
		HMIBinding.RackUI.sString20[2] := 'Solid_Red';
	END_IF;

	IF HMI.Rack7[24] >= 672 AND HMI.Rack7[24] <= 1080 THEN
		HMIBinding.RackUI.sString5[0] 	:= REAL_TO_STRING(HMI.Rack7[24]*0.1) ;
	ELSIF HMI.Rack7[24] < 672 THEN
		HMIBinding.RackUI.sString5[0]	:= '67.2';
	ELSE
		HMIBinding.RackUI.sString5[0]	:= '108';
	END_IF;
	HMIBinding.RackUI.sString20[5]		:= CONCAT(HMIBinding.RackUI.sString5[0],'(V)');

	IF (HMI.Rack7[21].2) THEN
		HMIBinding.RackUI.sString20[4] := 'Solid_Green';
	ELSE
		HMIBinding.RackUI.sString20[4] := 'Solid_Red';
	END_IF;

	IF HMI.Rack7[25] >= 672 AND HMI.Rack7[25] <= 1080 THEN
		HMIBinding.RackUI.sString5[0] 	:= REAL_TO_STRING(HMI.Rack7[25]*0.1) ;
	ELSIF HMI.Rack7[25] < 672 THEN
		HMIBinding.RackUI.sString5[0]	:= '67.2';
	ELSE
		HMIBinding.RackUI.sString5[0]	:= '108';
	END_IF;
	HMIBinding.RackUI.sString20[7]		:= CONCAT(HMIBinding.RackUI.sString5[0],'(V)');

	IF (HMI.Rack7[21].3) THEN
		HMIBinding.RackUI.sString20[6] := 'Solid_Green';
	ELSE
		HMIBinding.RackUI.sString20[6] := 'Solid_Red';
	END_IF;
	IF HMI.Rack7[26] >= 672 AND HMI.Rack7[26] <= 1080 THEN
		HMIBinding.RackUI.sString5[0] 	:= REAL_TO_STRING(HMI.Rack7[26]*0.1) ;
	ELSIF HMI.Rack7[26] < 672 THEN
		HMIBinding.RackUI.sString5[0]	:= '67.2';
	ELSE
		HMIBinding.RackUI.sString5[0]	:= '108';
	END_IF;
	HMIBinding.RackUI.sString20[9]		:= CONCAT(HMIBinding.RackUI.sString5[0],'(V)');

	IF (HMI.Rack7[21].4) THEN
		HMIBinding.RackUI.sString20[8] := 'Solid_Green';
	ELSE
		HMIBinding.RackUI.sString20[8] := 'Solid_Red';
	END_IF;
	IF HMI.Rack7[27] >= 672 AND HMI.Rack7[27] <= 1080 THEN
		HMIBinding.RackUI.sString5[0] 	:= REAL_TO_STRING(HMI.Rack7[27]*0.1) ;
	ELSIF HMI.Rack7[27] < 672 THEN
		HMIBinding.RackUI.sString5[0]	:= '67.2';
	ELSE
		HMIBinding.RackUI.sString5[0]	:= '108';
	END_IF;
	HMIBinding.RackUI.sString20[11]		:= CONCAT(HMIBinding.RackUI.sString5[0],'(V)');

	IF (HMI.Rack7[21].5) THEN
		HMIBinding.RackUI.sString20[10] := 'Solid_Green';
	ELSE
		HMIBinding.RackUI.sString20[10] := 'Solid_Red';
	END_IF;
	IF HMI.Rack7[28] >= 672 AND HMI.Rack7[28] <= 1080 THEN
		HMIBinding.RackUI.sString5[0] 	:= REAL_TO_STRING(HMI.Rack7[28]*0.1) ;
	ELSIF HMI.Rack7[28] < 672 THEN
		HMIBinding.RackUI.sString5[0]	:= '67.2';
	ELSE
		HMIBinding.RackUI.sString5[0]	:= '108';
	END_IF;
	HMIBinding.RackUI.sString20[13]		:= CONCAT(HMIBinding.RackUI.sString5[0],'(V)');

	IF (HMI.Rack7[21].6) THEN
		HMIBinding.RackUI.sString20[12] := 'Solid_Green';
	ELSE
		HMIBinding.RackUI.sString20[12] := 'Solid_Red';
	END_IF;

	(* Over Current *)
	IF HMI.Rack7[17].0 THEN
		HMIBinding.RackUI.sString20[14] 		:= 'Solid_Red';
	ELSIF HMI.Rack7[16].0 THEN
		HMIBinding.RackUI.sString20[14]			:= 'Solid_Orange';
	ELSIF HMI.Rack7[15].0 THEN
		HMIBinding.RackUI.sString20[14]			:= 'Solid_Yellow';
	ELSE
		HMIBinding.RackUI.sString20[14]			:= 'Solid_Green';
	END_IF;

	(* Over SOC *)
	IF HMI.Rack7[17].1 THEN
		HMIBinding.RackUI.sString20[15]			:= 'Solid_Red';
	ELSIF HMI.Rack7[16].1 THEN
		HMIBinding.RackUI.sString20[15]			:= 'Solid_Orange';
	ELSIF HMI.Rack7[15].1 THEN
		HMIBinding.RackUI.sString20[15]			:= 'Solid_Yellow';
	ELSE
		HMIBinding.RackUI.sString20[15] 			:= 'Solid_Green';
	END_IF;

	(* Under SOC *)
	IF HMI.Rack7[17].2 THEN
		HMIBinding.RackUI.sString20[16] 			:= 'Solid_Red';
	ELSIF HMI.Rack7[16].2 THEN
		HMIBinding.RackUI.sString20[16]  			:= 'Solid_Orange';
	ELSIF HMI.Rack7[15].2 THEN
		HMIBinding.RackUI.sString20[16] 			:= 'Solid_Yellow';
	ELSE
		HMIBinding.RackUI.sString20[16]			:= 'Solid_Green';
	END_IF;

	(* Over Voltage *)
	IF HMI.Rack7[17].3 THEN
		HMIBinding.RackUI.sString20[17]			:= 'Solid_Red';
	ELSIF HMI.Rack7[16].3 THEN
		HMIBinding.RackUI.sString20[17] 			:= 'Solid_Orange';
	ELSIF HMI.Rack7[15].3 THEN
		HMIBinding.RackUI.sString20[17] 			:= 'Solid_Yellow';
	ELSE
		HMIBinding.RackUI.sString20[17] 			:= 'Solid_Green';
	END_IF;

	(* Under Voltage *)
	IF HMI.Rack7[17].4 THEN
		HMIBinding.RackUI.sString20[18] 			:= 'Solid_Red';
	ELSIF HMI.Rack7[16].4 THEN
		HMIBinding.RackUI.sString20[18] 			:= 'Solid_Orange';
	ELSIF HMI.Rack7[15].4 THEN
		HMIBinding.RackUI.sString20[18] 			:= 'Solid_Yellow';
	ELSE
		HMIBinding.RackUI.sString20[18] 			:= 'Solid_Green';
	END_IF;

	(* Cell Over Voltage *)
	IF HMI.Rack7[17].5 THEN
		HMIBinding.RackUI.sString20[19] 			:= 'Solid_Red';
	ELSIF HMI.Rack7[16].5 THEN
		HMIBinding.RackUI.sString20[19] 			:= 'Solid_Orange';
	ELSIF HMI.Rack7[15].5 THEN
		HMIBinding.RackUI.sString20[19] 			:= 'Solid_Yellow';
	ELSE
		HMIBinding.RackUI.sString20[19] 			:= 'Solid_Green';
	END_IF;

	(* Cell Under Voltage *)
	IF HMI.Rack7[17].6 THEN
		HMIBinding.RackUI.sString20[20] 			:= 'Solid_Red';
	ELSIF HMI.Rack7[16].6 THEN
		HMIBinding.RackUI.sString20[20] 			:= 'Solid_Orange';
	ELSIF HMI.Rack7[15].6 THEN
		HMIBinding.RackUI.sString20[20] 			:= 'Solid_Yellow';
	ELSE
		HMIBinding.RackUI.sString20[20] 			:= 'Solid_Green';
	END_IF;

	(* Cell UnBalance Voltage *)
	IF HMI.Rack7[17].7 THEN
		HMIBinding.RackUI.sString20[21]			:= 'Solid_Red';
	ELSIF HMI.Rack7[16].7 THEN
		HMIBinding.RackUI.sString20[21] 			:= 'Solid_Orange';
	ELSIF HMI.Rack7[15].7 THEN
		HMIBinding.RackUI.sString20[21]			:= 'Solid_Yellow';
	ELSE
		HMIBinding.RackUI.sString20[21]			:= 'Solid_Green';
	END_IF;

	(* Discahrger Cell Over Temperature *)
	IF HMI.Rack7[17].8 THEN
		HMIBinding.RackUI.sString20[22] 			:= 'Solid_Red';
	ELSIF HMI.Rack7[16].8 THEN
		HMIBinding.RackUI.sString20[22] 			:= 'Solid_Orange';
	ELSIF HMI.Rack7[15].8 THEN
		HMIBinding.RackUI.sString20[22] 			:= 'Solid_Yellow';
	ELSE
		HMIBinding.RackUI.sString20[22] 			:= 'Solid_Green';
	END_IF;

	(* Charger Cell Over Temperature *)
	IF HMI.Rack7[17].9 THEN
		HMIBinding.RackUI.sString20[23] 			:= 'Solid_Red';
	ELSIF HMI.Rack7[16].9 THEN
		HMIBinding.RackUI.sString20[23] 			:= 'Solid_Orange';
	ELSIF HMI.Rack7[15].9 THEN
		HMIBinding.RackUI.sString20[23] 			:= 'Solid_Yellow';
	ELSE
		HMIBinding.RackUI.sString20[23] 			:= 'Solid_Green';
	END_IF;

	(* Discahrger Cell Under Temperature *)
	IF HMI.Rack7[17].10 THEN
		HMIBinding.RackUI.sString20[24] 			:= 'Solid_Red';
	ELSIF HMI.Rack7[16].10 THEN
		HMIBinding.RackUI.sString20[24] 			:= 'Solid_Orange';
	ELSIF HMI.Rack7[15].10 THEN
		HMIBinding.RackUI.sString20[24] 			:= 'Solid_Yellow';
	ELSE
		HMIBinding.RackUI.sString20[24] 			:= 'Solid_Green';
	END_IF;

	(* Charger Cell Under Temperature *)
	IF HMI.Rack7[17].11 THEN
		HMIBinding.RackUI.sString20[25] 		:= 'Solid_Red';
	ELSIF HMI.Rack7[16].11 THEN
		HMIBinding.RackUI.sString20[25]			:= 'Solid_Orange';
	ELSIF HMI.Rack7[15].11 THEN
		HMIBinding.RackUI.sString20[25]			:= 'Solid_Yellow';
	ELSE
		HMIBinding.RackUI.sString20[25]			:= 'Solid_Green';
	END_IF;

	(* Cell UnBalance Temperature *)
	IF HMI.Rack7[17].12 THEN
		HMIBinding.RackUI.sString20[26] 		:= 'Solid_Red';
	ELSIF HMI.Rack7[16].12 THEN
		HMIBinding.RackUI.sString20[26]			:= 'Solid_Orange';
	ELSIF HMI.Rack7[15].12 THEN
		HMIBinding.RackUI.sString20[26]			:= 'Solid_Yellow';
	ELSE
		HMIBinding.RackUI.sString20[26]			:= 'Solid_Green';
	END_IF;

	(* Internal COM *)
	IF HMI.Rack7[17].15 THEN
		HMIBinding.RackUI.sString20[27] 		:= 'Solid_Red';
	ELSE
		HMIBinding.RackUI.sString20[27]			:= 'Solid_Green';
	END_IF;

	(* External COM *)
	IF HMI.Rack7[17].0 THEN
		HMIBinding.RackUI.sString20[28] 		:= 'Solid_Red';
	ELSE
		HMIBinding.RackUI.sString20[28]			:= 'Solid_Green';
	END_IF;

	(* RelayWelding *)
	IF HMI.Rack7[18].1 THEN
		HMIBinding.RackUI.sString20[29] 		:= 'Solid_Red';
	ELSE
		HMIBinding.RackUI.sString20[29]			:= 'Solid_Green';
	END_IF;

	(* WaterLeak *)
	IF HMI.Rack7[18].2 THEN
		HMIBinding.RackUI.sString20[30] 		:= 'Solid_Red';
	ELSE
		HMIBinding.RackUI.sString20[30]			:= 'Solid_Green';
	END_IF;

	(* InsulationRegister *)
	IF HMI.Rack7[18].3 THEN
		HMIBinding.RackUI.sString20[31] 		:= 'Solid_Red';
	ELSE
		HMIBinding.RackUI.sString20[31]			:= 'Solid_Green';
	END_IF;

	(* MDSFuse *)
	IF HMI.Rack7[18].4 THEN
		HMIBinding.RackUI.sString20[32] 		:= 'Solid_Red';
	ELSE
		HMIBinding.RackUI.sString20[32]			:= 'Solid_Green';
	END_IF;

	(* CoolingRack *)
	IF HMI.Rack7[18].5 THEN
		HMIBinding.RackUI.sString20[33] 		:= 'Solid_Red';
	ELSE
		HMIBinding.RackUI.sString20[33]			:= 'Solid_Green';
	END_IF;

	(* DIO *)
	IF HMI.Rack7[19].0 THEN
		HMIBinding.RackUI.sString20[34] 		:= 'Solid_Red';
	ELSE
		HMIBinding.RackUI.sString20[34]			:= 'Solid_Green';
	END_IF;
	IF HMI.Rack7[19].1 THEN
		HMIBinding.RackUI.sString20[35] 		:= 'Solid_Red';
	ELSE
		HMIBinding.RackUI.sString20[35]			:= 'Solid_Green';
	END_IF;
	IF HMI.Rack7[19].2 THEN
		HMIBinding.RackUI.sString20[36] 		:= 'Solid_Red';
	ELSE
		HMIBinding.RackUI.sString20[36]			:= 'Solid_Green';
	END_IF;
	IF HMI.Rack7[20].2 THEN
		HMIBinding.RackUI.sString20[37] 		:= 'Solid_Red';
	ELSE
		HMIBinding.RackUI.sString20[37]			:= 'Solid_Green';
	END_IF;
	IF HMI.Rack7[20].4 THEN
		HMIBinding.RackUI.sString20[38] 		:= 'Solid_Red';
	ELSE
		HMIBinding.RackUI.sString20[38]			:= 'Solid_Green';
	END_IF;
	IF HMI.Rack7[20].5 THEN
		HMIBinding.RackUI.sString20[39] 		:= 'Solid_Red';
	ELSE
		HMIBinding.RackUI.sString20[39]			:= 'Solid_Green';
	END_IF;
END_ACTION
ACTION AtRack8UI :

	CASE HMI.Rack8[0] OF
		0:  HMIBinding.CommonUI.sString20[0] := 'NONE';
		1:  HMIBinding.CommonUI.sString20[0] := 'STANDBY';
		2:  HMIBinding.CommonUI.sString20[0] := 'RUN';
		3:  HMIBinding.CommonUI.sString20[0] := 'ALARM';
		4:  HMIBinding.CommonUI.sString20[0] := 'FAULT';
		5:  HMIBinding.CommonUI.sString20[0] := 'PROTECT';
	END_CASE;

	IF HMI.Rack8[1] >= 4700 AND HMI.Rack8[1] <= 7140 THEN
		HMIBinding.CommonUI.rReal[0]		:= UINT_TO_REAL(HMI.Rack8[1]) * 0.1 ;
	ELSIF HMI.Rack8[1] < 4700 THEN
		HMIBinding.CommonUI.rReal[0]		:= 470.0;
	ELSE
		HMIBinding.CommonUI.rReal[0]		:= 714.0;
	END_IF;
	HMIBinding.CommonUI.sString20[1]		:= REAL_TO_STRING((HMIBinding.CommonUI.rReal[0]-400)*0.675);
	HMIBinding.CommonUI.sString50[0]		:= CONCAT('[{"select":"#gauge3","spin":[',CONCAT(HMIBinding.CommonUI.sString20[1],',0,0]}]'));

	IF UINT_TO_INT(HMI.Rack8[2]) >= -3000 AND UINT_TO_INT(HMI.Rack8[2]) <= 3000 THEN
		HMIBinding.CommonUI.rReal[1] 			:= (UINT_TO_REAL(HMI.Rack8[2]) * 0.1) ;
	ELSIF UINT_TO_INT(HMI.Rack8[2]) < -3000 THEN
		HMIBinding.CommonUI.rReal[1]			:= -300;
	ELSE
		HMIBinding.CommonUI.rReal[1]			:= 300;
	END_IF;
	HMIBinding.CommonUI.sString20[2]		:= REAL_TO_STRING(HMIBinding.CommonUI.rReal[1]*0.27+135);
	HMIBinding.CommonUI.sString50[1]		:= CONCAT('[{"select":"#gauge4","spin":[',CONCAT(HMIBinding.CommonUI.sString20[2],',0,0]}]'));

	IF UINT_TO_INT(HMI.Rack8[3]) >= -50 AND UINT_TO_INT(HMI.Rack8[3]) <= 1050 THEN
		HMIBinding.CommonUI.rReal[2]		:= UINT_TO_REAL(HMI.Rack8[3]) * 0.1 ;
	ELSIF UINT_TO_INT(HMI.Rack8[3]) < -50 THEN
		HMIBinding.CommonUI.rReal[2]		:= -5;
	ELSE
		HMIBinding.CommonUI.rReal[2]		:= 105;
	END_IF;
	HMIBinding.CommonUI.sString20[3]		:= REAL_TO_STRING(HMIBinding.CommonUI.rReal[2]*2.7);
	HMIBinding.CommonUI.sString50[2]		:= CONCAT('[{"select":"#gauge1","spin":[',CONCAT(HMIBinding.CommonUI.sString20[3],',0,0]}]'));

	IF HMI.Rack8[4] >= 750 AND HMI.Rack8[4] <= 1000 THEN
		HMIBinding.CommonUI.rReal[3]		:= UINT_TO_REAL(HMI.Rack8[4]) * 0.1 ;
	ELSIF HMI.Rack8[4] < 750 THEN
		HMIBinding.CommonUI.rReal[3]		:= 75;
	ELSE
		HMIBinding.CommonUI.rReal[3]		:= 100;
	END_IF;
	HMIBinding.CommonUI.sString20[4]		:= REAL_TO_STRING(HMIBinding.CommonUI.rReal[3]*2.7);
	HMIBinding.CommonUI.sString50[3]		:= CONCAT('[{"select":"#gauge2","spin":[',CONCAT(HMIBinding.CommonUI.sString20[4],',0,0]}]'));

	IF HMI.Rack8[5] >= 2000 AND HMI.Rack8[5] <= 4500 THEN
		HMIBinding.CommonUI.rReal[4] 		:= UINT_TO_REAL(HMI.Rack8[5]) * 0.001 ;
	ELSIF	HMI.Rack8[5] < 2000 THEN
		HMIBinding.CommonUI.rReal[4]		:= 2;
	ELSE
		HMIBinding.CommonUI.rReal[4]		:= 4.5;
	END_IF;
	IF HMI.Rack8[6] >= 2000 AND HMI.Rack8[6] <= 4500 THEN
		HMIBinding.CommonUI.rReal[5]		:= UINT_TO_REAL(HMI.Rack8[6]) * 0.001 ;
	ELSIF	HMI.Rack8[6] < 2000 THEN
		HMIBinding.CommonUI.rReal[5]		:= 2;
	ELSE
		HMIBinding.CommonUI.rReal[5]		:= 4.5;
	END_IF;
	IF HMI.Rack8[7] >= 2000 AND HMI.Rack8[7] <= 4500 THEN
		HMIBinding.CommonUI.rReal[6]		:= UINT_TO_REAL(HMI.Rack8[7]) * 0.001 ;
	ELSIF	HMI.Rack8[7] < 2000 THEN
		HMIBinding.CommonUI.rReal[6]		:= 2;
	ELSE
		HMIBinding.CommonUI.rReal[6]		:= 4.5;
	END_IF;
	IF HMI.Rack8[8] >= 0 AND HMI.Rack8[8] <= 500 THEN
		HMIBinding.CommonUI.rReal[7] 		:= UINT_TO_REAL(HMI.Rack8[8]) * 0.001 ;
	ELSE
		HMIBinding.CommonUI.rReal[7] 		:= 0.5;
	END_IF;
	IF UINT_TO_INT(HMI.Rack8[9]) >= -300 AND UINT_TO_INT(HMI.Rack8[9]) <= 1000 THEN
		HMIBinding.CommonUI.rReal[8] 		:= UINT_TO_REAL(HMI.Rack8[9]) * 0.1 ;
	ELSIF	UINT_TO_INT(HMI.Rack8[9]) < -300 THEN
		HMIBinding.CommonUI.rReal[8] 		:= -30;
	ELSE
		HMIBinding.CommonUI.rReal[8] 		:= 100;
	END_IF;
	IF UINT_TO_INT(HMI.Rack8[10]) >= -300 AND UINT_TO_INT(HMI.Rack8[10]) <= 1000 THEN
		HMIBinding.CommonUI.rReal[9]		:= UINT_TO_REAL(HMI.Rack8[10]) * 0.1 ;
	ELSIF	UINT_TO_INT(HMI.Rack8[10]) < -300 THEN
		HMIBinding.CommonUI.rReal[9]		:= -30;
	ELSE
		HMIBinding.CommonUI.rReal[9]		:= 100;
	END_IF;
	IF UINT_TO_INT(HMI.Rack8[11]) >= -300 AND UINT_TO_INT(HMI.Rack8[11]) <= 1000 THEN
		HMIBinding.CommonUI.rReal[10]		:= UINT_TO_REAL(HMI.Rack8[11]) * 0.1 ;
	ELSIF	UINT_TO_INT(HMI.Rack8[11]) < -300 THEN
		HMIBinding.CommonUI.rReal[10]		:= -30;
	ELSE
		HMIBinding.CommonUI.rReal[10]		:= 100;
	END_IF;
	IF HMI.Rack8[12] >= 0 AND HMI.Rack8[12] <= 100 THEN
		HMIBinding.CommonUI.rReal[11] 		:= UINT_TO_REAL(HMI.Rack8[12]) * 0.1 ;
	ELSE
		HMIBinding.CommonUI.rReal[11]		:= 10;
	END_IF;

	IF (HMI.Rack8[13] AND 16#00ff) >= 1 AND (HMI.Rack8[13] AND 16#00ff) <= 164 THEN
		HMIBinding.CommonUI.sString5[0]		:= UINT_TO_STRING((HMI.Rack8[13] AND 16#00ff)) ;
	ELSIF (HMI.Rack8[13] AND 16#00ff) < 1 THEN
		HMIBinding.CommonUI.sString5[0]		:= '1';
	ELSE
		HMIBinding.CommonUI.sString5[0]		:= '164';
	END_IF;
	IF (HMI.Rack8[13]  /  16#0100) >= 1 AND (HMI.Rack8[13]  /  16#0100) <= 164 THEN
		HMIBinding.CommonUI.sString5[1] 		:= UINT_TO_STRING(HMI.Rack8[13]  /  16#0100) ;
	ELSIF (HMI.Rack8[13]  /  16#0100) < 1 THEN
		HMIBinding.CommonUI.sString5[1]		:= '1';
	ELSE
		HMIBinding.CommonUI.sString5[1]		:= '164';
	END_IF;
	HMIBinding.CommonUI.sString20[5]		:= CONCAT(HMIBinding.CommonUI.sString5[0],'(C)');
	HMIBinding.CommonUI.sString20[6]		:= CONCAT(HMIBinding.CommonUI.sString5[1],'(C)');

	IF (HMI.Rack8[14] AND 16#00ff) >= 1 AND (HMI.Rack8[14] AND 16#00ff) <= 164 THEN
		HMIBinding.CommonUI.sString5[0]		:= UINT_TO_STRING((HMI.Rack8[14] AND 16#00ff)) ;
	ELSIF (HMI.Rack8[14] AND 16#00ff) < 1 THEN
		HMIBinding.CommonUI.sString5[0]		:= '1';
	ELSE
		HMIBinding.CommonUI.sString5[0]		:= '164';
	END_IF;
	IF (HMI.Rack8[14]  /  16#0100) >= 1 AND (HMI.Rack8[14]  /  16#0100) <= 164 THEN
		HMIBinding.CommonUI.sString5[1] 		:= UINT_TO_STRING(HMI.Rack8[14]  /  16#0100) ;
	ELSIF (HMI.Rack8[14]  /  16#0100) < 1 THEN
		HMIBinding.CommonUI.sString5[1]		:= '1';
	ELSE
		HMIBinding.CommonUI.sString5[1]		:= '164';
	END_IF;
	HMIBinding.CommonUI.sString20[7]		:= CONCAT(HMIBinding.CommonUI.sString5[0],'(C)');
	HMIBinding.CommonUI.sString20[8]		:= CONCAT(HMIBinding.CommonUI.sString5[1],'(C)');

	IF HMI.Rack8[22] >= 672 AND HMI.Rack8[22] <= 1080 THEN
		HMIBinding.RackUI.sString5[0] 	:= REAL_TO_STRING(HMI.Rack8[22]*0.1) ;
	ELSIF HMI.Rack8[22] < 672 THEN
		HMIBinding.RackUI.sString5[0]	:= '67.2';
	ELSE
		HMIBinding.RackUI.sString5[0]	:= '108';
	END_IF;
	HMIBinding.RackUI.sString20[1]		:= CONCAT(HMIBinding.RackUI.sString5[0],'(V)');

	IF (HMI.Rack8[21].0) THEN
		HMIBinding.RackUI.sString20[0] := 'Solid_Green';
	ELSE
		HMIBinding.RackUI.sString20[0] := 'Solid_Red';
	END_IF;
	IF HMI.Rack8[23] >= 672 AND HMI.Rack8[23] <= 1080 THEN
		HMIBinding.RackUI.sString5[0] 	:= REAL_TO_STRING(HMI.Rack8[23]*0.1) ;
	ELSIF HMI.Rack8[23] < 672 THEN
		HMIBinding.RackUI.sString5[0]	:= '67.2';
	ELSE
		HMIBinding.RackUI.sString5[0]	:= '108';
	END_IF;
	HMIBinding.RackUI.sString20[3]		:= CONCAT(HMIBinding.RackUI.sString5[0],'(V)');

	IF (HMI.Rack8[21].1) THEN
		HMIBinding.RackUI.sString20[2] := 'Solid_Green';
	ELSE
		HMIBinding.RackUI.sString20[2] := 'Solid_Red';
	END_IF;

	IF HMI.Rack8[24] >= 672 AND HMI.Rack8[24] <= 1080 THEN
		HMIBinding.RackUI.sString5[0] 	:= REAL_TO_STRING(HMI.Rack8[24]*0.1) ;
	ELSIF HMI.Rack8[24] < 672 THEN
		HMIBinding.RackUI.sString5[0]	:= '67.2';
	ELSE
		HMIBinding.RackUI.sString5[0]	:= '108';
	END_IF;
	HMIBinding.RackUI.sString20[5]		:= CONCAT(HMIBinding.RackUI.sString5[0],'(V)');

	IF (HMI.Rack8[21].2) THEN
		HMIBinding.RackUI.sString20[4] := 'Solid_Green';
	ELSE
		HMIBinding.RackUI.sString20[4] := 'Solid_Red';
	END_IF;

	IF HMI.Rack8[25] >= 672 AND HMI.Rack8[25] <= 1080 THEN
		HMIBinding.RackUI.sString5[0] 	:= REAL_TO_STRING(HMI.Rack8[25]*0.1) ;
	ELSIF HMI.Rack8[25] < 672 THEN
		HMIBinding.RackUI.sString5[0]	:= '67.2';
	ELSE
		HMIBinding.RackUI.sString5[0]	:= '108';
	END_IF;
	HMIBinding.RackUI.sString20[7]		:= CONCAT(HMIBinding.RackUI.sString5[0],'(V)');

	IF (HMI.Rack8[21].3) THEN
		HMIBinding.RackUI.sString20[6] := 'Solid_Green';
	ELSE
		HMIBinding.RackUI.sString20[6] := 'Solid_Red';
	END_IF;
	IF HMI.Rack8[26] >= 672 AND HMI.Rack8[26] <= 1080 THEN
		HMIBinding.RackUI.sString5[0] 	:= REAL_TO_STRING(HMI.Rack8[26]*0.1) ;
	ELSIF HMI.Rack8[26] < 672 THEN
		HMIBinding.RackUI.sString5[0]	:= '67.2';
	ELSE
		HMIBinding.RackUI.sString5[0]	:= '108';
	END_IF;
	HMIBinding.RackUI.sString20[9]		:= CONCAT(HMIBinding.RackUI.sString5[0],'(V)');

	IF (HMI.Rack8[21].4) THEN
		HMIBinding.RackUI.sString20[8] := 'Solid_Green';
	ELSE
		HMIBinding.RackUI.sString20[8] := 'Solid_Red';
	END_IF;
	IF HMI.Rack8[27] >= 672 AND HMI.Rack8[27] <= 1080 THEN
		HMIBinding.RackUI.sString5[0] 	:= REAL_TO_STRING(HMI.Rack8[27]*0.1) ;
	ELSIF HMI.Rack8[27] < 672 THEN
		HMIBinding.RackUI.sString5[0]	:= '67.2';
	ELSE
		HMIBinding.RackUI.sString5[0]	:= '108';
	END_IF;
	HMIBinding.RackUI.sString20[11]		:= CONCAT(HMIBinding.RackUI.sString5[0],'(V)');

	IF (HMI.Rack8[21].5) THEN
		HMIBinding.RackUI.sString20[10] := 'Solid_Green';
	ELSE
		HMIBinding.RackUI.sString20[10] := 'Solid_Red';
	END_IF;
	IF HMI.Rack8[28] >= 672 AND HMI.Rack8[28] <= 1080 THEN
		HMIBinding.RackUI.sString5[0] 	:= REAL_TO_STRING(HMI.Rack8[28]*0.1) ;
	ELSIF HMI.Rack8[28] < 672 THEN
		HMIBinding.RackUI.sString5[0]	:= '67.2';
	ELSE
		HMIBinding.RackUI.sString5[0]	:= '108';
	END_IF;
	HMIBinding.RackUI.sString20[13]		:= CONCAT(HMIBinding.RackUI.sString5[0],'(V)');

	IF (HMI.Rack8[21].6) THEN
		HMIBinding.RackUI.sString20[12] := 'Solid_Green';
	ELSE
		HMIBinding.RackUI.sString20[12] := 'Solid_Red';
	END_IF;

	(* Over Current *)
	IF HMI.Rack8[17].0 THEN
		HMIBinding.RackUI.sString20[14] 		:= 'Solid_Red';
	ELSIF HMI.Rack8[16].0 THEN
		HMIBinding.RackUI.sString20[14]			:= 'Solid_Orange';
	ELSIF HMI.Rack8[15].0 THEN
		HMIBinding.RackUI.sString20[14]			:= 'Solid_Yellow';
	ELSE
		HMIBinding.RackUI.sString20[14]			:= 'Solid_Green';
	END_IF;

	(* Over SOC *)
	IF HMI.Rack8[17].1 THEN
		HMIBinding.RackUI.sString20[15]			:= 'Solid_Red';
	ELSIF HMI.Rack8[16].1 THEN
		HMIBinding.RackUI.sString20[15]			:= 'Solid_Orange';
	ELSIF HMI.Rack8[15].1 THEN
		HMIBinding.RackUI.sString20[15]			:= 'Solid_Yellow';
	ELSE
		HMIBinding.RackUI.sString20[15] 			:= 'Solid_Green';
	END_IF;

	(* Under SOC *)
	IF HMI.Rack8[17].2 THEN
		HMIBinding.RackUI.sString20[16] 			:= 'Solid_Red';
	ELSIF HMI.Rack8[16].2 THEN
		HMIBinding.RackUI.sString20[16]  			:= 'Solid_Orange';
	ELSIF HMI.Rack8[15].2 THEN
		HMIBinding.RackUI.sString20[16] 			:= 'Solid_Yellow';
	ELSE
		HMIBinding.RackUI.sString20[16]			:= 'Solid_Green';
	END_IF;

	(* Over Voltage *)
	IF HMI.Rack8[17].3 THEN
		HMIBinding.RackUI.sString20[17]			:= 'Solid_Red';
	ELSIF HMI.Rack8[16].3 THEN
		HMIBinding.RackUI.sString20[17] 			:= 'Solid_Orange';
	ELSIF HMI.Rack8[15].3 THEN
		HMIBinding.RackUI.sString20[17] 			:= 'Solid_Yellow';
	ELSE
		HMIBinding.RackUI.sString20[17] 			:= 'Solid_Green';
	END_IF;

	(* Under Voltage *)
	IF HMI.Rack8[17].4 THEN
		HMIBinding.RackUI.sString20[18] 			:= 'Solid_Red';
	ELSIF HMI.Rack8[16].4 THEN
		HMIBinding.RackUI.sString20[18] 			:= 'Solid_Orange';
	ELSIF HMI.Rack8[15].4 THEN
		HMIBinding.RackUI.sString20[18] 			:= 'Solid_Yellow';
	ELSE
		HMIBinding.RackUI.sString20[18] 			:= 'Solid_Green';
	END_IF;

	(* Cell Over Voltage *)
	IF HMI.Rack8[17].5 THEN
		HMIBinding.RackUI.sString20[19] 			:= 'Solid_Red';
	ELSIF HMI.Rack8[16].5 THEN
		HMIBinding.RackUI.sString20[19] 			:= 'Solid_Orange';
	ELSIF HMI.Rack8[15].5 THEN
		HMIBinding.RackUI.sString20[19] 			:= 'Solid_Yellow';
	ELSE
		HMIBinding.RackUI.sString20[19] 			:= 'Solid_Green';
	END_IF;

	(* Cell Under Voltage *)
	IF HMI.Rack8[17].6 THEN
		HMIBinding.RackUI.sString20[20] 			:= 'Solid_Red';
	ELSIF HMI.Rack8[16].6 THEN
		HMIBinding.RackUI.sString20[20] 			:= 'Solid_Orange';
	ELSIF HMI.Rack8[15].6 THEN
		HMIBinding.RackUI.sString20[20] 			:= 'Solid_Yellow';
	ELSE
		HMIBinding.RackUI.sString20[20] 			:= 'Solid_Green';
	END_IF;

	(* Cell UnBalance Voltage *)
	IF HMI.Rack8[17].7 THEN
		HMIBinding.RackUI.sString20[21]			:= 'Solid_Red';
	ELSIF HMI.Rack8[16].7 THEN
		HMIBinding.RackUI.sString20[21] 			:= 'Solid_Orange';
	ELSIF HMI.Rack8[15].7 THEN
		HMIBinding.RackUI.sString20[21]			:= 'Solid_Yellow';
	ELSE
		HMIBinding.RackUI.sString20[21]			:= 'Solid_Green';
	END_IF;

	(* Discahrger Cell Over Temperature *)
	IF HMI.Rack8[17].8 THEN
		HMIBinding.RackUI.sString20[22] 			:= 'Solid_Red';
	ELSIF HMI.Rack8[16].8 THEN
		HMIBinding.RackUI.sString20[22] 			:= 'Solid_Orange';
	ELSIF HMI.Rack8[15].8 THEN
		HMIBinding.RackUI.sString20[22] 			:= 'Solid_Yellow';
	ELSE
		HMIBinding.RackUI.sString20[22] 			:= 'Solid_Green';
	END_IF;

	(* Charger Cell Over Temperature *)
	IF HMI.Rack8[17].9 THEN
		HMIBinding.RackUI.sString20[23] 			:= 'Solid_Red';
	ELSIF HMI.Rack8[16].9 THEN
		HMIBinding.RackUI.sString20[23] 			:= 'Solid_Orange';
	ELSIF HMI.Rack8[15].9 THEN
		HMIBinding.RackUI.sString20[23] 			:= 'Solid_Yellow';
	ELSE
		HMIBinding.RackUI.sString20[23] 			:= 'Solid_Green';
	END_IF;

	(* Discahrger Cell Under Temperature *)
	IF HMI.Rack8[17].10 THEN
		HMIBinding.RackUI.sString20[24] 			:= 'Solid_Red';
	ELSIF HMI.Rack8[16].10 THEN
		HMIBinding.RackUI.sString20[24] 			:= 'Solid_Orange';
	ELSIF HMI.Rack8[15].10 THEN
		HMIBinding.RackUI.sString20[24] 			:= 'Solid_Yellow';
	ELSE
		HMIBinding.RackUI.sString20[24] 			:= 'Solid_Green';
	END_IF;

	(* Charger Cell Under Temperature *)
	IF HMI.Rack8[17].11 THEN
		HMIBinding.RackUI.sString20[25] 		:= 'Solid_Red';
	ELSIF HMI.Rack8[16].11 THEN
		HMIBinding.RackUI.sString20[25]			:= 'Solid_Orange';
	ELSIF HMI.Rack8[15].11 THEN
		HMIBinding.RackUI.sString20[25]			:= 'Solid_Yellow';
	ELSE
		HMIBinding.RackUI.sString20[25]			:= 'Solid_Green';
	END_IF;

	(* Cell UnBalance Temperature *)
	IF HMI.Rack8[17].12 THEN
		HMIBinding.RackUI.sString20[26] 		:= 'Solid_Red';
	ELSIF HMI.Rack8[16].12 THEN
		HMIBinding.RackUI.sString20[26]			:= 'Solid_Orange';
	ELSIF HMI.Rack8[15].12 THEN
		HMIBinding.RackUI.sString20[26]			:= 'Solid_Yellow';
	ELSE
		HMIBinding.RackUI.sString20[26]			:= 'Solid_Green';
	END_IF;

	(* Internal COM *)
	IF HMI.Rack8[17].15 THEN
		HMIBinding.RackUI.sString20[27] 		:= 'Solid_Red';
	ELSE
		HMIBinding.RackUI.sString20[27]			:= 'Solid_Green';
	END_IF;

	(* External COM *)
	IF HMI.Rack8[17].0 THEN
		HMIBinding.RackUI.sString20[28] 		:= 'Solid_Red';
	ELSE
		HMIBinding.RackUI.sString20[28]			:= 'Solid_Green';
	END_IF;

	(* RelayWelding *)
	IF HMI.Rack8[18].1 THEN
		HMIBinding.RackUI.sString20[29] 		:= 'Solid_Red';
	ELSE
		HMIBinding.RackUI.sString20[29]			:= 'Solid_Green';
	END_IF;

	(* WaterLeak *)
	IF HMI.Rack8[18].2 THEN
		HMIBinding.RackUI.sString20[30] 		:= 'Solid_Red';
	ELSE
		HMIBinding.RackUI.sString20[30]			:= 'Solid_Green';
	END_IF;

	(* InsulationRegister *)
	IF HMI.Rack8[18].3 THEN
		HMIBinding.RackUI.sString20[31] 		:= 'Solid_Red';
	ELSE
		HMIBinding.RackUI.sString20[31]			:= 'Solid_Green';
	END_IF;

	(* MDSFuse *)
	IF HMI.Rack8[18].4 THEN
		HMIBinding.RackUI.sString20[32] 		:= 'Solid_Red';
	ELSE
		HMIBinding.RackUI.sString20[32]			:= 'Solid_Green';
	END_IF;

	(* CoolingRack *)
	IF HMI.Rack8[18].5 THEN
		HMIBinding.RackUI.sString20[33] 		:= 'Solid_Red';
	ELSE
		HMIBinding.RackUI.sString20[33]			:= 'Solid_Green';
	END_IF;

	(* DIO *)
	IF HMI.Rack8[19].0 THEN
		HMIBinding.RackUI.sString20[34] 		:= 'Solid_Red';
	ELSE
		HMIBinding.RackUI.sString20[34]			:= 'Solid_Green';
	END_IF;
	IF HMI.Rack8[19].1 THEN
		HMIBinding.RackUI.sString20[35] 		:= 'Solid_Red';
	ELSE
		HMIBinding.RackUI.sString20[35]			:= 'Solid_Green';
	END_IF;
	IF HMI.Rack8[19].2 THEN
		HMIBinding.RackUI.sString20[36] 		:= 'Solid_Red';
	ELSE
		HMIBinding.RackUI.sString20[36]			:= 'Solid_Green';
	END_IF;
	IF HMI.Rack8[20].2 THEN
		HMIBinding.RackUI.sString20[37] 		:= 'Solid_Red';
	ELSE
		HMIBinding.RackUI.sString20[37]			:= 'Solid_Green';
	END_IF;
	IF HMI.Rack8[20].4 THEN
		HMIBinding.RackUI.sString20[38] 		:= 'Solid_Red';
	ELSE
		HMIBinding.RackUI.sString20[38]			:= 'Solid_Green';
	END_IF;
	IF HMI.Rack8[20].5 THEN
		HMIBinding.RackUI.sString20[39] 		:= 'Solid_Red';
	ELSE
		HMIBinding.RackUI.sString20[39]			:= 'Solid_Green';
	END_IF;
END_ACTION
ACTION AtRack9UI :

	CASE HMI.Rack9[0] OF
		0:  HMIBinding.CommonUI.sString20[0] := 'NONE';
		1:  HMIBinding.CommonUI.sString20[0] := 'STANDBY';
		2:  HMIBinding.CommonUI.sString20[0] := 'RUN';
		3:  HMIBinding.CommonUI.sString20[0] := 'ALARM';
		4:  HMIBinding.CommonUI.sString20[0] := 'FAULT';
		5:  HMIBinding.CommonUI.sString20[0] := 'PROTECT';
	END_CASE;

	IF HMI.Rack9[1] >= 4700 AND HMI.Rack9[1] <= 7140 THEN
		HMIBinding.CommonUI.rReal[0]		:= UINT_TO_REAL(HMI.Rack9[1]) * 0.1 ;
	ELSIF HMI.Rack9[1] < 4700 THEN
		HMIBinding.CommonUI.rReal[0]		:= 470.0;
	ELSE
		HMIBinding.CommonUI.rReal[0]		:= 714.0;
	END_IF;
	HMIBinding.CommonUI.sString20[1]		:= REAL_TO_STRING((HMIBinding.CommonUI.rReal[0]-400)*0.675);
	HMIBinding.CommonUI.sString50[0]		:= CONCAT('[{"select":"#gauge3","spin":[',CONCAT(HMIBinding.CommonUI.sString20[1],',0,0]}]'));

	IF UINT_TO_INT(HMI.Rack9[2]) >= -3000 AND UINT_TO_INT(HMI.Rack9[2]) <= 3000 THEN
		HMIBinding.CommonUI.rReal[1] 			:= (UINT_TO_REAL(HMI.Rack9[2]) * 0.1) ;
	ELSIF UINT_TO_INT(HMI.Rack9[2]) < -3000 THEN
		HMIBinding.CommonUI.rReal[1]			:= -300;
	ELSE
		HMIBinding.CommonUI.rReal[1]			:= 300;
	END_IF;
	HMIBinding.CommonUI.sString20[2]		:= REAL_TO_STRING(HMIBinding.CommonUI.rReal[1]*0.27+135);
	HMIBinding.CommonUI.sString50[1]		:= CONCAT('[{"select":"#gauge4","spin":[',CONCAT(HMIBinding.CommonUI.sString20[2],',0,0]}]'));

	IF UINT_TO_INT(HMI.Rack9[3]) >= -50 AND UINT_TO_INT(HMI.Rack9[3]) <= 1050 THEN
		HMIBinding.CommonUI.rReal[2]		:= UINT_TO_REAL(HMI.Rack9[3]) * 0.1 ;
	ELSIF UINT_TO_INT(HMI.Rack9[3]) < -50 THEN
		HMIBinding.CommonUI.rReal[2]		:= -5;
	ELSE
		HMIBinding.CommonUI.rReal[2]		:= 105;
	END_IF;
	HMIBinding.CommonUI.sString20[3]		:= REAL_TO_STRING(HMIBinding.CommonUI.rReal[2]*2.7);
	HMIBinding.CommonUI.sString50[2]		:= CONCAT('[{"select":"#gauge1","spin":[',CONCAT(HMIBinding.CommonUI.sString20[3],',0,0]}]'));

	IF HMI.Rack9[4] >= 750 AND HMI.Rack9[4] <= 1000 THEN
		HMIBinding.CommonUI.rReal[3]		:= UINT_TO_REAL(HMI.Rack9[4]) * 0.1 ;
	ELSIF HMI.Rack9[4] < 750 THEN
		HMIBinding.CommonUI.rReal[3]		:= 75;
	ELSE
		HMIBinding.CommonUI.rReal[3]		:= 100;
	END_IF;
	HMIBinding.CommonUI.sString20[4]		:= REAL_TO_STRING(HMIBinding.CommonUI.rReal[3]*2.7);
	HMIBinding.CommonUI.sString50[3]		:= CONCAT('[{"select":"#gauge2","spin":[',CONCAT(HMIBinding.CommonUI.sString20[4],',0,0]}]'));

	IF HMI.Rack9[5] >= 2000 AND HMI.Rack9[5] <= 4500 THEN
		HMIBinding.CommonUI.rReal[4] 		:= UINT_TO_REAL(HMI.Rack9[5]) * 0.001 ;
	ELSIF	HMI.Rack9[5] < 2000 THEN
		HMIBinding.CommonUI.rReal[4]		:= 2;
	ELSE
		HMIBinding.CommonUI.rReal[4]		:= 4.5;
	END_IF;
	IF HMI.Rack9[6] >= 2000 AND HMI.Rack9[6] <= 4500 THEN
		HMIBinding.CommonUI.rReal[5]		:= UINT_TO_REAL(HMI.Rack9[6]) * 0.001 ;
	ELSIF	HMI.Rack9[6] < 2000 THEN
		HMIBinding.CommonUI.rReal[5]		:= 2;
	ELSE
		HMIBinding.CommonUI.rReal[5]		:= 4.5;
	END_IF;
	IF HMI.Rack9[7] >= 2000 AND HMI.Rack9[7] <= 4500 THEN
		HMIBinding.CommonUI.rReal[6]		:= UINT_TO_REAL(HMI.Rack9[7]) * 0.001 ;
	ELSIF	HMI.Rack9[7] < 2000 THEN
		HMIBinding.CommonUI.rReal[6]		:= 2;
	ELSE
		HMIBinding.CommonUI.rReal[6]		:= 4.5;
	END_IF;
	IF HMI.Rack9[8] >= 0 AND HMI.Rack9[8] <= 500 THEN
		HMIBinding.CommonUI.rReal[7] 		:= UINT_TO_REAL(HMI.Rack9[8]) * 0.001 ;
	ELSE
		HMIBinding.CommonUI.rReal[7] 		:= 0.5;
	END_IF;
	IF UINT_TO_INT(HMI.Rack9[9]) >= -300 AND UINT_TO_INT(HMI.Rack9[9]) <= 1000 THEN
		HMIBinding.CommonUI.rReal[8] 		:= UINT_TO_REAL(HMI.Rack9[9]) * 0.1 ;
	ELSIF	UINT_TO_INT(HMI.Rack9[9]) < -300 THEN
		HMIBinding.CommonUI.rReal[8] 		:= -30;
	ELSE
		HMIBinding.CommonUI.rReal[8] 		:= 100;
	END_IF;
	IF UINT_TO_INT(HMI.Rack9[10]) >= -300 AND UINT_TO_INT(HMI.Rack9[10]) <= 1000 THEN
		HMIBinding.CommonUI.rReal[9]		:= UINT_TO_REAL(HMI.Rack9[10]) * 0.1 ;
	ELSIF	UINT_TO_INT(HMI.Rack9[10]) < -300 THEN
		HMIBinding.CommonUI.rReal[9]		:= -30;
	ELSE
		HMIBinding.CommonUI.rReal[9]		:= 100;
	END_IF;
	IF UINT_TO_INT(HMI.Rack9[11]) >= -300 AND UINT_TO_INT(HMI.Rack9[11]) <= 1000 THEN
		HMIBinding.CommonUI.rReal[10]		:= UINT_TO_REAL(HMI.Rack9[11]) * 0.1 ;
	ELSIF	UINT_TO_INT(HMI.Rack9[11]) < -300 THEN
		HMIBinding.CommonUI.rReal[10]		:= -30;
	ELSE
		HMIBinding.CommonUI.rReal[10]		:= 100;
	END_IF;
	IF HMI.Rack9[12] >= 0 AND HMI.Rack9[12] <= 100 THEN
		HMIBinding.CommonUI.rReal[11] 		:= UINT_TO_REAL(HMI.Rack9[12]) * 0.1 ;
	ELSE
		HMIBinding.CommonUI.rReal[11]		:= 10;
	END_IF;

	IF (HMI.Rack9[13] AND 16#00ff) >= 1 AND (HMI.Rack9[13] AND 16#00ff) <= 164 THEN
		HMIBinding.CommonUI.sString5[0]		:= UINT_TO_STRING((HMI.Rack9[13] AND 16#00ff)) ;
	ELSIF (HMI.Rack9[13] AND 16#00ff) < 1 THEN
		HMIBinding.CommonUI.sString5[0]		:= '1';
	ELSE
		HMIBinding.CommonUI.sString5[0]		:= '164';
	END_IF;
	IF (HMI.Rack9[13]  /  16#0100) >= 1 AND (HMI.Rack9[13]  /  16#0100) <= 164 THEN
		HMIBinding.CommonUI.sString5[1] 		:= UINT_TO_STRING(HMI.Rack9[13]  /  16#0100) ;
	ELSIF (HMI.Rack9[13]  /  16#0100) < 1 THEN
		HMIBinding.CommonUI.sString5[1]		:= '1';
	ELSE
		HMIBinding.CommonUI.sString5[1]		:= '164';
	END_IF;
	HMIBinding.CommonUI.sString20[5]		:= CONCAT(HMIBinding.CommonUI.sString5[0],'(C)');
	HMIBinding.CommonUI.sString20[6]		:= CONCAT(HMIBinding.CommonUI.sString5[1],'(C)');

	IF (HMI.Rack9[14] AND 16#00ff) >= 1 AND (HMI.Rack9[14] AND 16#00ff) <= 164 THEN
		HMIBinding.CommonUI.sString5[0]		:= UINT_TO_STRING((HMI.Rack9[14] AND 16#00ff)) ;
	ELSIF (HMI.Rack9[14] AND 16#00ff) < 1 THEN
		HMIBinding.CommonUI.sString5[0]		:= '1';
	ELSE
		HMIBinding.CommonUI.sString5[0]		:= '164';
	END_IF;
	IF (HMI.Rack9[14]  /  16#0100) >= 1 AND (HMI.Rack9[14]  /  16#0100) <= 164 THEN
		HMIBinding.CommonUI.sString5[1] 		:= UINT_TO_STRING(HMI.Rack9[14]  /  16#0100) ;
	ELSIF (HMI.Rack9[14]  /  16#0100) < 1 THEN
		HMIBinding.CommonUI.sString5[1]		:= '1';
	ELSE
		HMIBinding.CommonUI.sString5[1]		:= '164';
	END_IF;
	HMIBinding.CommonUI.sString20[7]		:= CONCAT(HMIBinding.CommonUI.sString5[0],'(C)');
	HMIBinding.CommonUI.sString20[8]		:= CONCAT(HMIBinding.CommonUI.sString5[1],'(C)');

	IF HMI.Rack9[22] >= 672 AND HMI.Rack9[22] <= 1080 THEN
		HMIBinding.RackUI.sString5[0] 	:= REAL_TO_STRING(HMI.Rack9[22]*0.1) ;
	ELSIF HMI.Rack9[22] < 672 THEN
		HMIBinding.RackUI.sString5[0]	:= '67.2';
	ELSE
		HMIBinding.RackUI.sString5[0]	:= '108';
	END_IF;
	HMIBinding.RackUI.sString20[1]		:= CONCAT(HMIBinding.RackUI.sString5[0],'(V)');

	IF (HMI.Rack9[21].0) THEN
		HMIBinding.RackUI.sString20[0] := 'Solid_Green';
	ELSE
		HMIBinding.RackUI.sString20[0] := 'Solid_Red';
	END_IF;
	IF HMI.Rack9[23] >= 672 AND HMI.Rack9[23] <= 1080 THEN
		HMIBinding.RackUI.sString5[0] 	:= REAL_TO_STRING(HMI.Rack9[23]*0.1) ;
	ELSIF HMI.Rack9[23] < 672 THEN
		HMIBinding.RackUI.sString5[0]	:= '67.2';
	ELSE
		HMIBinding.RackUI.sString5[0]	:= '108';
	END_IF;
	HMIBinding.RackUI.sString20[3]		:= CONCAT(HMIBinding.RackUI.sString5[0],'(V)');

	IF (HMI.Rack9[21].1) THEN
		HMIBinding.RackUI.sString20[2] := 'Solid_Green';
	ELSE
		HMIBinding.RackUI.sString20[2] := 'Solid_Red';
	END_IF;

	IF HMI.Rack9[24] >= 672 AND HMI.Rack9[24] <= 1080 THEN
		HMIBinding.RackUI.sString5[0] 	:= REAL_TO_STRING(HMI.Rack9[24]*0.1) ;
	ELSIF HMI.Rack9[24] < 672 THEN
		HMIBinding.RackUI.sString5[0]	:= '67.2';
	ELSE
		HMIBinding.RackUI.sString5[0]	:= '108';
	END_IF;
	HMIBinding.RackUI.sString20[5]		:= CONCAT(HMIBinding.RackUI.sString5[0],'(V)');

	IF (HMI.Rack9[21].2) THEN
		HMIBinding.RackUI.sString20[4] := 'Solid_Green';
	ELSE
		HMIBinding.RackUI.sString20[4] := 'Solid_Red';
	END_IF;

	IF HMI.Rack9[25] >= 672 AND HMI.Rack9[25] <= 1080 THEN
		HMIBinding.RackUI.sString5[0] 	:= REAL_TO_STRING(HMI.Rack9[25]*0.1) ;
	ELSIF HMI.Rack9[25] < 672 THEN
		HMIBinding.RackUI.sString5[0]	:= '67.2';
	ELSE
		HMIBinding.RackUI.sString5[0]	:= '108';
	END_IF;
	HMIBinding.RackUI.sString20[7]		:= CONCAT(HMIBinding.RackUI.sString5[0],'(V)');

	IF (HMI.Rack9[21].3) THEN
		HMIBinding.RackUI.sString20[6] := 'Solid_Green';
	ELSE
		HMIBinding.RackUI.sString20[6] := 'Solid_Red';
	END_IF;
	IF HMI.Rack9[26] >= 672 AND HMI.Rack9[26] <= 1080 THEN
		HMIBinding.RackUI.sString5[0] 	:= REAL_TO_STRING(HMI.Rack9[26]*0.1) ;
	ELSIF HMI.Rack9[26] < 672 THEN
		HMIBinding.RackUI.sString5[0]	:= '67.2';
	ELSE
		HMIBinding.RackUI.sString5[0]	:= '108';
	END_IF;
	HMIBinding.RackUI.sString20[9]		:= CONCAT(HMIBinding.RackUI.sString5[0],'(V)');

	IF (HMI.Rack9[21].4) THEN
		HMIBinding.RackUI.sString20[8] := 'Solid_Green';
	ELSE
		HMIBinding.RackUI.sString20[8] := 'Solid_Red';
	END_IF;
	IF HMI.Rack9[27] >= 672 AND HMI.Rack9[27] <= 1080 THEN
		HMIBinding.RackUI.sString5[0] 	:= REAL_TO_STRING(HMI.Rack9[27]*0.1) ;
	ELSIF HMI.Rack9[27] < 672 THEN
		HMIBinding.RackUI.sString5[0]	:= '67.2';
	ELSE
		HMIBinding.RackUI.sString5[0]	:= '108';
	END_IF;
	HMIBinding.RackUI.sString20[11]		:= CONCAT(HMIBinding.RackUI.sString5[0],'(V)');

	IF (HMI.Rack9[21].5) THEN
		HMIBinding.RackUI.sString20[10] := 'Solid_Green';
	ELSE
		HMIBinding.RackUI.sString20[10] := 'Solid_Red';
	END_IF;
	IF HMI.Rack9[28] >= 672 AND HMI.Rack9[28] <= 1080 THEN
		HMIBinding.RackUI.sString5[0] 	:= REAL_TO_STRING(HMI.Rack9[28]*0.1) ;
	ELSIF HMI.Rack9[28] < 672 THEN
		HMIBinding.RackUI.sString5[0]	:= '67.2';
	ELSE
		HMIBinding.RackUI.sString5[0]	:= '108';
	END_IF;
	HMIBinding.RackUI.sString20[13]		:= CONCAT(HMIBinding.RackUI.sString5[0],'(V)');

	IF (HMI.Rack9[21].6) THEN
		HMIBinding.RackUI.sString20[12] := 'Solid_Green';
	ELSE
		HMIBinding.RackUI.sString20[12] := 'Solid_Red';
	END_IF;

	(* Over Current *)
	IF HMI.Rack9[17].0 THEN
		HMIBinding.RackUI.sString20[14] 		:= 'Solid_Red';
	ELSIF HMI.Rack9[16].0 THEN
		HMIBinding.RackUI.sString20[14]			:= 'Solid_Orange';
	ELSIF HMI.Rack9[15].0 THEN
		HMIBinding.RackUI.sString20[14]			:= 'Solid_Yellow';
	ELSE
		HMIBinding.RackUI.sString20[14]			:= 'Solid_Green';
	END_IF;

	(* Over SOC *)
	IF HMI.Rack9[17].1 THEN
		HMIBinding.RackUI.sString20[15]			:= 'Solid_Red';
	ELSIF HMI.Rack9[16].1 THEN
		HMIBinding.RackUI.sString20[15]			:= 'Solid_Orange';
	ELSIF HMI.Rack9[15].1 THEN
		HMIBinding.RackUI.sString20[15]			:= 'Solid_Yellow';
	ELSE
		HMIBinding.RackUI.sString20[15] 			:= 'Solid_Green';
	END_IF;

	(* Under SOC *)
	IF HMI.Rack9[17].2 THEN
		HMIBinding.RackUI.sString20[16] 			:= 'Solid_Red';
	ELSIF HMI.Rack9[16].2 THEN
		HMIBinding.RackUI.sString20[16]  			:= 'Solid_Orange';
	ELSIF HMI.Rack9[15].2 THEN
		HMIBinding.RackUI.sString20[16] 			:= 'Solid_Yellow';
	ELSE
		HMIBinding.RackUI.sString20[16]			:= 'Solid_Green';
	END_IF;

	(* Over Voltage *)
	IF HMI.Rack9[17].3 THEN
		HMIBinding.RackUI.sString20[17]			:= 'Solid_Red';
	ELSIF HMI.Rack9[16].3 THEN
		HMIBinding.RackUI.sString20[17] 			:= 'Solid_Orange';
	ELSIF HMI.Rack9[15].3 THEN
		HMIBinding.RackUI.sString20[17] 			:= 'Solid_Yellow';
	ELSE
		HMIBinding.RackUI.sString20[17] 			:= 'Solid_Green';
	END_IF;

	(* Under Voltage *)
	IF HMI.Rack9[17].4 THEN
		HMIBinding.RackUI.sString20[18] 			:= 'Solid_Red';
	ELSIF HMI.Rack9[16].4 THEN
		HMIBinding.RackUI.sString20[18] 			:= 'Solid_Orange';
	ELSIF HMI.Rack9[15].4 THEN
		HMIBinding.RackUI.sString20[18] 			:= 'Solid_Yellow';
	ELSE
		HMIBinding.RackUI.sString20[18] 			:= 'Solid_Green';
	END_IF;

	(* Cell Over Voltage *)
	IF HMI.Rack9[17].5 THEN
		HMIBinding.RackUI.sString20[19] 			:= 'Solid_Red';
	ELSIF HMI.Rack9[16].5 THEN
		HMIBinding.RackUI.sString20[19] 			:= 'Solid_Orange';
	ELSIF HMI.Rack9[15].5 THEN
		HMIBinding.RackUI.sString20[19] 			:= 'Solid_Yellow';
	ELSE
		HMIBinding.RackUI.sString20[19] 			:= 'Solid_Green';
	END_IF;

	(* Cell Under Voltage *)
	IF HMI.Rack9[17].6 THEN
		HMIBinding.RackUI.sString20[20] 			:= 'Solid_Red';
	ELSIF HMI.Rack9[16].6 THEN
		HMIBinding.RackUI.sString20[20] 			:= 'Solid_Orange';
	ELSIF HMI.Rack9[15].6 THEN
		HMIBinding.RackUI.sString20[20] 			:= 'Solid_Yellow';
	ELSE
		HMIBinding.RackUI.sString20[20] 			:= 'Solid_Green';
	END_IF;

	(* Cell UnBalance Voltage *)
	IF HMI.Rack9[17].7 THEN
		HMIBinding.RackUI.sString20[21]			:= 'Solid_Red';
	ELSIF HMI.Rack9[16].7 THEN
		HMIBinding.RackUI.sString20[21] 			:= 'Solid_Orange';
	ELSIF HMI.Rack9[15].7 THEN
		HMIBinding.RackUI.sString20[21]			:= 'Solid_Yellow';
	ELSE
		HMIBinding.RackUI.sString20[21]			:= 'Solid_Green';
	END_IF;

	(* Discahrger Cell Over Temperature *)
	IF HMI.Rack9[17].8 THEN
		HMIBinding.RackUI.sString20[22] 			:= 'Solid_Red';
	ELSIF HMI.Rack9[16].8 THEN
		HMIBinding.RackUI.sString20[22] 			:= 'Solid_Orange';
	ELSIF HMI.Rack9[15].8 THEN
		HMIBinding.RackUI.sString20[22] 			:= 'Solid_Yellow';
	ELSE
		HMIBinding.RackUI.sString20[22] 			:= 'Solid_Green';
	END_IF;

	(* Charger Cell Over Temperature *)
	IF HMI.Rack9[17].9 THEN
		HMIBinding.RackUI.sString20[23] 			:= 'Solid_Red';
	ELSIF HMI.Rack9[16].9 THEN
		HMIBinding.RackUI.sString20[23] 			:= 'Solid_Orange';
	ELSIF HMI.Rack9[15].9 THEN
		HMIBinding.RackUI.sString20[23] 			:= 'Solid_Yellow';
	ELSE
		HMIBinding.RackUI.sString20[23] 			:= 'Solid_Green';
	END_IF;

	(* Discahrger Cell Under Temperature *)
	IF HMI.Rack9[17].10 THEN
		HMIBinding.RackUI.sString20[24] 			:= 'Solid_Red';
	ELSIF HMI.Rack9[16].10 THEN
		HMIBinding.RackUI.sString20[24] 			:= 'Solid_Orange';
	ELSIF HMI.Rack9[15].10 THEN
		HMIBinding.RackUI.sString20[24] 			:= 'Solid_Yellow';
	ELSE
		HMIBinding.RackUI.sString20[24] 			:= 'Solid_Green';
	END_IF;

	(* Charger Cell Under Temperature *)
	IF HMI.Rack9[17].11 THEN
		HMIBinding.RackUI.sString20[25] 		:= 'Solid_Red';
	ELSIF HMI.Rack9[16].11 THEN
		HMIBinding.RackUI.sString20[25]			:= 'Solid_Orange';
	ELSIF HMI.Rack9[15].11 THEN
		HMIBinding.RackUI.sString20[25]			:= 'Solid_Yellow';
	ELSE
		HMIBinding.RackUI.sString20[25]			:= 'Solid_Green';
	END_IF;

	(* Cell UnBalance Temperature *)
	IF HMI.Rack9[17].12 THEN
		HMIBinding.RackUI.sString20[26] 		:= 'Solid_Red';
	ELSIF HMI.Rack9[16].12 THEN
		HMIBinding.RackUI.sString20[26]			:= 'Solid_Orange';
	ELSIF HMI.Rack9[15].12 THEN
		HMIBinding.RackUI.sString20[26]			:= 'Solid_Yellow';
	ELSE
		HMIBinding.RackUI.sString20[26]			:= 'Solid_Green';
	END_IF;

	(* Internal COM *)
	IF HMI.Rack9[17].15 THEN
		HMIBinding.RackUI.sString20[27] 		:= 'Solid_Red';
	ELSE
		HMIBinding.RackUI.sString20[27]			:= 'Solid_Green';
	END_IF;

	(* External COM *)
	IF HMI.Rack9[17].0 THEN
		HMIBinding.RackUI.sString20[28] 		:= 'Solid_Red';
	ELSE
		HMIBinding.RackUI.sString20[28]			:= 'Solid_Green';
	END_IF;

	(* RelayWelding *)
	IF HMI.Rack9[18].1 THEN
		HMIBinding.RackUI.sString20[29] 		:= 'Solid_Red';
	ELSE
		HMIBinding.RackUI.sString20[29]			:= 'Solid_Green';
	END_IF;

	(* WaterLeak *)
	IF HMI.Rack9[18].2 THEN
		HMIBinding.RackUI.sString20[30] 		:= 'Solid_Red';
	ELSE
		HMIBinding.RackUI.sString20[30]			:= 'Solid_Green';
	END_IF;

	(* InsulationRegister *)
	IF HMI.Rack9[18].3 THEN
		HMIBinding.RackUI.sString20[31] 		:= 'Solid_Red';
	ELSE
		HMIBinding.RackUI.sString20[31]			:= 'Solid_Green';
	END_IF;

	(* MDSFuse *)
	IF HMI.Rack9[18].4 THEN
		HMIBinding.RackUI.sString20[32] 		:= 'Solid_Red';
	ELSE
		HMIBinding.RackUI.sString20[32]			:= 'Solid_Green';
	END_IF;

	(* CoolingRack *)
	IF HMI.Rack9[18].5 THEN
		HMIBinding.RackUI.sString20[33] 		:= 'Solid_Red';
	ELSE
		HMIBinding.RackUI.sString20[33]			:= 'Solid_Green';
	END_IF;

	(* DIO *)
	IF HMI.Rack9[19].0 THEN
		HMIBinding.RackUI.sString20[34] 		:= 'Solid_Red';
	ELSE
		HMIBinding.RackUI.sString20[34]			:= 'Solid_Green';
	END_IF;
	IF HMI.Rack9[19].1 THEN
		HMIBinding.RackUI.sString20[35] 		:= 'Solid_Red';
	ELSE
		HMIBinding.RackUI.sString20[35]			:= 'Solid_Green';
	END_IF;
	IF HMI.Rack9[19].2 THEN
		HMIBinding.RackUI.sString20[36] 		:= 'Solid_Red';
	ELSE
		HMIBinding.RackUI.sString20[36]			:= 'Solid_Green';
	END_IF;
	IF HMI.Rack9[20].2 THEN
		HMIBinding.RackUI.sString20[37] 		:= 'Solid_Red';
	ELSE
		HMIBinding.RackUI.sString20[37]			:= 'Solid_Green';
	END_IF;
	IF HMI.Rack9[20].4 THEN
		HMIBinding.RackUI.sString20[38] 		:= 'Solid_Red';
	ELSE
		HMIBinding.RackUI.sString20[38]			:= 'Solid_Green';
	END_IF;
	IF HMI.Rack9[20].5 THEN
		HMIBinding.RackUI.sString20[39] 		:= 'Solid_Red';
	ELSE
		HMIBinding.RackUI.sString20[39]			:= 'Solid_Green';
	END_IF;
END_ACTION
ACTION AtRack10UI :

	CASE HMI.Rack10[0] OF
		0:  HMIBinding.CommonUI.sString20[0] := 'NONE';
		1:  HMIBinding.CommonUI.sString20[0] := 'STANDBY';
		2:  HMIBinding.CommonUI.sString20[0] := 'RUN';
		3:  HMIBinding.CommonUI.sString20[0] := 'ALARM';
		4:  HMIBinding.CommonUI.sString20[0] := 'FAULT';
		5:  HMIBinding.CommonUI.sString20[0] := 'PROTECT';
	END_CASE;

	IF HMI.Rack10[1] >= 4700 AND HMI.Rack10[1] <= 7140 THEN
		HMIBinding.CommonUI.rReal[0]		:= UINT_TO_REAL(HMI.Rack10[1]) * 0.1 ;
	ELSIF HMI.Rack10[1] < 4700 THEN
		HMIBinding.CommonUI.rReal[0]		:= 470.0;
	ELSE
		HMIBinding.CommonUI.rReal[0]		:= 714.0;
	END_IF;
	HMIBinding.CommonUI.sString20[1]		:= REAL_TO_STRING((HMIBinding.CommonUI.rReal[0]-400)*0.675);
	HMIBinding.CommonUI.sString50[0]		:= CONCAT('[{"select":"#gauge3","spin":[',CONCAT(HMIBinding.CommonUI.sString20[1],',0,0]}]'));

	IF UINT_TO_INT(HMI.Rack10[2]) >= -3000 AND UINT_TO_INT(HMI.Rack10[2]) <= 3000 THEN
		HMIBinding.CommonUI.rReal[1] 			:= (UINT_TO_REAL(HMI.Rack10[2]) * 0.1) ;
	ELSIF UINT_TO_INT(HMI.Rack10[2]) < -3000 THEN
		HMIBinding.CommonUI.rReal[1]			:= -300;
	ELSE
		HMIBinding.CommonUI.rReal[1]			:= 300;
	END_IF;
	HMIBinding.CommonUI.sString20[2]		:= REAL_TO_STRING(HMIBinding.CommonUI.rReal[1]*0.27+135);
	HMIBinding.CommonUI.sString50[1]		:= CONCAT('[{"select":"#gauge4","spin":[',CONCAT(HMIBinding.CommonUI.sString20[2],',0,0]}]'));

	IF UINT_TO_INT(HMI.Rack10[3]) >= -50 AND UINT_TO_INT(HMI.Rack10[3]) <= 1050 THEN
		HMIBinding.CommonUI.rReal[2]		:= UINT_TO_REAL(HMI.Rack10[3]) * 0.1 ;
	ELSIF UINT_TO_INT(HMI.Rack10[3]) < -50 THEN
		HMIBinding.CommonUI.rReal[2]		:= -5;
	ELSE
		HMIBinding.CommonUI.rReal[2]		:= 105;
	END_IF;
	HMIBinding.CommonUI.sString20[3]		:= REAL_TO_STRING(HMIBinding.CommonUI.rReal[2]*2.7);
	HMIBinding.CommonUI.sString50[2]		:= CONCAT('[{"select":"#gauge1","spin":[',CONCAT(HMIBinding.CommonUI.sString20[3],',0,0]}]'));

	IF HMI.Rack10[4] >= 750 AND HMI.Rack10[4] <= 1000 THEN
		HMIBinding.CommonUI.rReal[3]		:= UINT_TO_REAL(HMI.Rack10[4]) * 0.1 ;
	ELSIF HMI.Rack10[4] < 750 THEN
		HMIBinding.CommonUI.rReal[3]		:= 75;
	ELSE
		HMIBinding.CommonUI.rReal[3]		:= 100;
	END_IF;
	HMIBinding.CommonUI.sString20[4]		:= REAL_TO_STRING(HMIBinding.CommonUI.rReal[3]*2.7);
	HMIBinding.CommonUI.sString50[3]		:= CONCAT('[{"select":"#gauge2","spin":[',CONCAT(HMIBinding.CommonUI.sString20[4],',0,0]}]'));

	IF HMI.Rack10[5] >= 2000 AND HMI.Rack10[5] <= 4500 THEN
		HMIBinding.CommonUI.rReal[4] 		:= UINT_TO_REAL(HMI.Rack10[5]) * 0.001 ;
	ELSIF	HMI.Rack10[5] < 2000 THEN
		HMIBinding.CommonUI.rReal[4]		:= 2;
	ELSE
		HMIBinding.CommonUI.rReal[4]		:= 4.5;
	END_IF;
	IF HMI.Rack10[6] >= 2000 AND HMI.Rack10[6] <= 4500 THEN
		HMIBinding.CommonUI.rReal[5]		:= UINT_TO_REAL(HMI.Rack10[6]) * 0.001 ;
	ELSIF	HMI.Rack10[6] < 2000 THEN
		HMIBinding.CommonUI.rReal[5]		:= 2;
	ELSE
		HMIBinding.CommonUI.rReal[5]		:= 4.5;
	END_IF;
	IF HMI.Rack10[7] >= 2000 AND HMI.Rack10[7] <= 4500 THEN
		HMIBinding.CommonUI.rReal[6]		:= UINT_TO_REAL(HMI.Rack10[7]) * 0.001 ;
	ELSIF	HMI.Rack10[7] < 2000 THEN
		HMIBinding.CommonUI.rReal[6]		:= 2;
	ELSE
		HMIBinding.CommonUI.rReal[6]		:= 4.5;
	END_IF;
	IF HMI.Rack10[8] >= 0 AND HMI.Rack10[8] <= 500 THEN
		HMIBinding.CommonUI.rReal[7] 		:= UINT_TO_REAL(HMI.Rack10[8]) * 0.001 ;
	ELSE
		HMIBinding.CommonUI.rReal[7] 		:= 0.5;
	END_IF;
	IF UINT_TO_INT(HMI.Rack10[9]) >= -300 AND UINT_TO_INT(HMI.Rack10[9]) <= 1000 THEN
		HMIBinding.CommonUI.rReal[8] 		:= UINT_TO_REAL(HMI.Rack10[9]) * 0.1 ;
	ELSIF	UINT_TO_INT(HMI.Rack10[9]) < -300 THEN
		HMIBinding.CommonUI.rReal[8] 		:= -30;
	ELSE
		HMIBinding.CommonUI.rReal[8] 		:= 100;
	END_IF;
	IF UINT_TO_INT(HMI.Rack10[10]) >= -300 AND UINT_TO_INT(HMI.Rack10[10]) <= 1000 THEN
		HMIBinding.CommonUI.rReal[9]		:= UINT_TO_REAL(HMI.Rack10[10]) * 0.1 ;
	ELSIF	UINT_TO_INT(HMI.Rack10[10]) < -300 THEN
		HMIBinding.CommonUI.rReal[9]		:= -30;
	ELSE
		HMIBinding.CommonUI.rReal[9]		:= 100;
	END_IF;
	IF UINT_TO_INT(HMI.Rack10[11]) >= -300 AND UINT_TO_INT(HMI.Rack10[11]) <= 1000 THEN
		HMIBinding.CommonUI.rReal[10]		:= UINT_TO_REAL(HMI.Rack10[11]) * 0.1 ;
	ELSIF	UINT_TO_INT(HMI.Rack10[11]) < -300 THEN
		HMIBinding.CommonUI.rReal[10]		:= -30;
	ELSE
		HMIBinding.CommonUI.rReal[10]		:= 100;
	END_IF;
	IF HMI.Rack10[12] >= 0 AND HMI.Rack10[12] <= 100 THEN
		HMIBinding.CommonUI.rReal[11] 		:= UINT_TO_REAL(HMI.Rack10[12]) * 0.1 ;
	ELSE
		HMIBinding.CommonUI.rReal[11]		:= 10;
	END_IF;
